LIN {X 0,Y 530.553,Z 620.523,A -85,B 0,C 180,E1 -4403.152,E2 -4403.152} C_VEL
LIN {X 0,Y 530.515,Z 626.199,A -85,B 0,C 180,E1 -4404.678,E2 -4404.678} C_VEL
LIN {X 0,Y 530.497,Z 630.318,A -85,B 0,C 180,E1 -4406.201,E2 -4406.201} C_VEL
LIN {X 0,Y 530.409,Z 633.003,A -85,B 0,C 180,E1 -4407.721,E2 -4407.721} C_VEL
LIN {X 0,Y 530.341,Z 634.333,A -85,B 0,C 180,E1 -4409.24,E2 -4409.24} C_VEL
LIN {X 0,Y 530.341,Z 634.334,A -85,B 0,C 180,E1 -4410.758,E2 -4410.758} C_VEL
LIN {X 0,Y 530.409,Z 633.003,A -85,B 0,C 180,E1 -4412.277,E2 -4412.277} C_VEL
LIN {X 0,Y 530.496,Z 630.318,A -85,B 0,C 180,E1 -4413.797,E2 -4413.797} C_VEL
LIN {X 0,Y 530.514,Z 626.204,A -85,B 0,C 180,E1 -4415.32,E2 -4415.32} C_VEL
LIN {X 0,Y 530.572,Z 620.532,A -85,B 0,C 180,E1 -4416.846,E2 -4416.846} C_VEL
LIN {X 0,Y 530.708,Z 614.132,A -85,B 0,C 180,E1 -4418.183,E2 -4418.183} C_VEL
LIN {X 0,Y 530.928,Z 606.18,A -85,B 0,C 180,E1 -4419.523,E2 -4419.523} C_VEL
LIN {X 0,Y 531.129,Z 597.86,A -85,B 0,C 180,E1 -4420.675,E2 -4420.675} C_VEL
LIN {X 0,Y 531.452,Z 587.362,A -85,B 0,C 180,E1 -4421.878,E2 -4421.878} C_VEL
LIN {X 0,Y 531.717,Z 576.66,A -85,B 0,C 180,E1 -4422.887,E2 -4422.887} C_VEL
LIN {X 0,Y 532.08,Z 564.113,A -85,B 0,C 180,E1 -4423.85,E2 -4423.85} C_VEL
LIN {X 0,Y 532.482,Z 551.655,A -85,B 0,C 180,E1 -4424.62,E2 -4424.62} C_VEL
LIN {X 0,Y 532.81,Z 537.728,A -85,B 0,C 180,E1 -4425.295,E2 -4425.295} C_VEL
LIN {X 0,Y 533.063,Z 523.832,A -85,B 0,C 180,E1 -4425.796,E2 -4425.796} C_VEL
LIN {X 0,Y 533.146,Z 510.218,A -85,B 0,C 180,E1 -4426.137,E2 -4426.137} C_VEL
LIN {X 0,Y 531.159,Z 499.764,A -85,B 0,C 180,E1 -4426.378,E2 -4426.378} C_VEL
LIN {X 0,Y 531.354,Z 487.006,A -85,B 0,C 180,E1 -4428.907,E2 -4428.907} C_VEL
LIN {X 0,Y 531.562,Z 471.4,A -85,B 0,C 180,E1 -4431.993,E2 -4431.993} C_VEL
LIN {X 0,Y 531.756,Z 457.556,A -85,B 0,C 180,E1 -4434.81,E2 -4434.81} C_VEL
LIN {X 0,Y 532.001,Z 444.494,A -85,B 0,C 180,E1 -4437.539,E2 -4437.539} C_VEL
LIN {X 0,Y 532.22,Z 430.626,A -85,B 0,C 180,E1 -4440.5,E2 -4440.5} C_VEL
LIN {X 0,Y 532.488,Z 417.378,A -85,B 0,C 180,E1 -4443.437,E2 -4443.437} C_VEL
LIN {X 0,Y 532.955,Z 402.449,A -85,B 0,C 180,E1 -4446.868,E2 -4446.868} C_VEL
LIN {X 0,Y 533.188,Z 395.134,A -85,B 0,C 180,E1 -4448.606,E2 -4448.606} C_VEL
LIN {X 0,Y 532.7,Z 391.02,A -85,B 0,C 180,E1 -4449.645,E2 -4449.645} C_VEL
LIN {X 0,Y 531.002,Z 382.968,A -85,B 0,C 180,E1 -4451.821,E2 -4451.821} C_VEL
LIN {X 0,Y 530.982,Z 382.967,A -85,B 0,C 180,E1 -4454.546,E2 -4454.546} C_VEL
LIN {X 0,Y 530.991,Z 382.971,A -85,B 0,C 180,E1 -4457.831,E2 -4457.831} C_VEL
LIN {X 0,Y 530.998,Z 382.963,A -85,B 0,C 180,E1 -4460.558,E2 -4460.558} C_VEL
LIN {X 0,Y 530.967,Z 382.972,A -85,B 0,C 180,E1 -4463.841,E2 -4463.841} C_VEL
LIN {X 0,Y 530.991,Z 382.964,A -85,B 0,C 180,E1 -4466.493,E2 -4466.493} C_VEL
LIN {X 0,Y 530.973,Z 382.97,A -85,B 0,C 180,E1 -4469.353,E2 -4469.353} C_VEL
LIN {X 0,Y 531.008,Z 382.962,A -85,B 0,C 180,E1 -4472.404,E2 -4472.404} C_VEL
LIN {X 0,Y 530.998,Z 382.964,A -85,B 0,C 180,E1 -4474.942,E2 -4474.942} C_VEL
LIN {X 0,Y 530.961,Z 382.969,A -85,B 0,C 180,E1 -4478.246,E2 -4478.246} C_VEL
LIN {X 0,Y 530.987,Z 382.964,A -85,B 0,C 180,E1 -4480.677,E2 -4480.677} C_VEL
LIN {X 0,Y 530.984,Z 382.967,A -85,B 0,C 180,E1 -4483.071,E2 -4483.071} C_VEL
LIN {X 0,Y 531.03,Z 382.966,A -85,B 0,C 180,E1 -4485.436,E2 -4485.436} C_VEL
LIN {X 0,Y 531.036,Z 382.958,A -85,B 0,C 180,E1 -4488.55,E2 -4488.55} C_VEL
LIN {X 0,Y 531.05,Z 382.962,A -85,B 0,C 180,E1 -4491.63,E2 -4491.63} C_VEL
LIN {X 0,Y 531.115,Z 382.949,A -85,B 0,C 180,E1 -4494.685,E2 -4494.685} C_VEL
LIN {X 0,Y 531.13,Z 382.951,A -85,B 0,C 180,E1 -4497.725,E2 -4497.725} C_VEL
LIN {X 0,Y 531.146,Z 382.945,A -85,B 0,C 180,E1 -4500.758,E2 -4500.758} C_VEL
LIN {X 0,Y 531.101,Z 382.953,A -85,B 0,C 180,E1 -4503.034,E2 -4503.034} C_VEL
LIN {X 0,Y 531.075,Z 382.954,A -85,B 0,C 180,E1 -4506.077,E2 -4506.077} C_VEL
LIN {X 0,Y 531.027,Z 382.965,A -85,B 0,C 180,E1 -4509.138,E2 -4509.138} C_VEL
LIN {X 0,Y 531.031,Z 382.959,A -85,B 0,C 180,E1 -4512.225,E2 -4512.225} C_VEL
LIN {X 0,Y 530.987,Z 382.971,A -85,B 0,C 180,E1 -4515.35,E2 -4515.35} C_VEL
LIN {X 0,Y 531.007,Z 382.966,A -85,B 0,C 180,E1 -4517.723,E2 -4517.723} C_VEL
LIN {X 0,Y 530.993,Z 382.967,A -85,B 0,C 180,E1 -4520.938,E2 -4520.938} C_VEL
LIN {X 0,Y 530.971,Z 382.966,A -85,B 0,C 180,E1 -4524.225,E2 -4524.225} C_VEL
LIN {X 0,Y 531.004,Z 382.964,A -85,B 0,C 180,E1 -4526.744,E2 -4526.744} C_VEL
LIN {X 0,Y 530.975,Z 382.971,A -85,B 0,C 180,E1 -4529.323,E2 -4529.323} C_VEL
LIN {X 0,Y 530.973,Z 382.966,A -85,B 0,C 180,E1 -4532.104,E2 -4532.104} C_VEL
LIN {X 0,Y 530.984,Z 382.969,A -85,B 0,C 180,E1 -4534.855,E2 -4534.855} C_VEL
LIN {X 0,Y 530.961,Z 382.972,A -85,B 0,C 180,E1 -4537.509,E2 -4537.509} C_VEL
LIN {X 0,Y 530.979,Z 382.966,A -85,B 0,C 180,E1 -4540.434,E2 -4540.434} C_VEL
LIN {X 0,Y 530.963,Z 382.972,A -85,B 0,C 180,E1 -4543.495,E2 -4543.495} C_VEL
LIN {X 0,Y 530.96,Z 382.971,A -85,B 0,C 180,E1 -4543.578,E2 -4543.578} C_VEL
LIN {X 0,Y 530.286,Z 383.052,A -85,B 0,C 180,E1 -4544.212,E2 -4544.212} C_VEL
LIN {X 0,Y 527.437,Z 383.412,A -85,B 0,C 180,E1 -4545.24,E2 -4545.24} C_VEL
LIN {X 0,Y 525.032,Z 383.714,A -85,B 0,C 180,E1 -4546.069,E2 -4546.069} C_VEL
LIN {X 0,Y 524,Z 383.84,A -85,B 0,C 180,E1 -4546.708,E2 -4546.708} C_VEL
LIN {X 0,Y 523.915,Z 383.85,A -85,B 0,C 180,E1 -4546.925,E2 -4546.925} C_VEL
LIN {X 0,Y 523.975,Z 383.838,A -85,B 0,C 180,E1 -4549.925,E2 -4549.925} C_VEL
LIN {X 0,Y 523.909,Z 383.852,A -85,B 0,C 180,E1 -4552.87,E2 -4552.87} C_VEL
LIN {X 0,Y 523.943,Z 383.843,A -85,B 0,C 180,E1 -4555.712,E2 -4555.712} C_VEL
LIN {X 0,Y 523.93,Z 383.845,A -85,B 0,C 180,E1 -4558.458,E2 -4558.458} C_VEL
LIN {X 0,Y 523.939,Z 383.847,A -85,B 0,C 180,E1 -4561.127,E2 -4561.127} C_VEL
LIN {X 0,Y 523.985,Z 383.837,A -85,B 0,C 180,E1 -4563.981,E2 -4563.981} C_VEL
LIN {X 0,Y 523.927,Z 383.845,A -85,B 0,C 180,E1 -4566.271,E2 -4566.271} C_VEL
LIN {X 0,Y 523.947,Z 383.848,A -85,B 0,C 180,E1 -4568.768,E2 -4568.768} C_VEL
LIN {X 0,Y 523.951,Z 383.845,A -85,B 0,C 180,E1 -4571.222,E2 -4571.222} C_VEL
LIN {X 0,Y 523.923,Z 383.845,A -85,B 0,C 180,E1 -4573.639,E2 -4573.639} C_VEL
LIN {X 0,Y 523.811,Z 383.865,A -85,B 0,C 180,E1 -4576.026,E2 -4576.026} C_VEL
LIN {X 0,Y 523.644,Z 383.885,A -85,B 0,C 180,E1 -4578.454,E2 -4578.454} C_VEL
LIN {X 0,Y 523.539,Z 383.897,A -85,B 0,C 180,E1 -4579.389,E2 -4579.389} C_VEL
LIN {X 0,Y 525.473,Z 393.055,A -85,B 0,C 180,E1 -4579.696,E2 -4579.696} C_VEL
LIN {X 0,Y 525.341,Z 405.307,A -85,B 0,C 180,E1 -4580.131,E2 -4580.131} C_VEL
LIN {X 0,Y 525.11,Z 416.338,A -85,B 0,C 180,E1 -4580.662,E2 -4580.662} C_VEL
LIN {X 0,Y 524.825,Z 427.193,A -85,B 0,C 180,E1 -4581.336,E2 -4581.336} C_VEL
LIN {X 0,Y 524.474,Z 438.244,A -85,B 0,C 180,E1 -4582.203,E2 -4582.203} C_VEL
LIN {X 0,Y 524.21,Z 447.187,A -85,B 0,C 180,E1 -4583.071,E2 -4583.071} C_VEL
LIN {X 0,Y 524.089,Z 455.344,A -85,B 0,C 180,E1 -4584.036,E2 -4584.036} C_VEL
LIN {X 0,Y 523.822,Z 463.291,A -85,B 0,C 180,E1 -4585.191,E2 -4585.191} C_VEL
LIN {X 0,Y 523.672,Z 470.642,A -85,B 0,C 180,E1 -4586.539,E2 -4586.539} C_VEL
LIN {X 0,Y 523.47,Z 475.563,A -85,B 0,C 180,E1 -4587.693,E2 -4587.693} C_VEL
LIN {X 0,Y 523.457,Z 479.343,A -85,B 0,C 180,E1 -4588.847,E2 -4588.847} C_VEL
LIN {X 0,Y 523.299,Z 482.152,A -85,B 0,C 180,E1 -4590.001,E2 -4590.001} C_VEL
LIN {X 0,Y 523.3,Z 484.416,A -85,B 0,C 180,E1 -4591.54,E2 -4591.54} C_VEL
LIN {X 0,Y 523.39,Z 485.162,A -85,B 0,C 180,E1 -4593.08,E2 -4593.08} C_VEL
LIN {X 0,Y 523.433,Z 484.927,A -85,B 0,C 180,E1 -4593.85,E2 -4593.85} C_VEL
LIN {X 0,Y 523.397,Z 483.363,A -85,B 0,C 180,E1 -4595.394,E2 -4595.394} C_VEL
LIN {X 0,Y 523.432,Z 481.253,A -85,B 0,C 180,E1 -4596.492,E2 -4596.492} C_VEL
LIN {X 0,Y 523.451,Z 477.911,A -85,B 0,C 180,E1 -4597.717,E2 -4597.717} C_VEL
LIN {X 0,Y 523.576,Z 473.64,A -85,B 0,C 180,E1 -4598.881,E2 -4598.881} C_VEL
LIN {X 0,Y 523.721,Z 467.117,A -85,B 0,C 180,E1 -4600.243,E2 -4600.243} C_VEL
LIN {X 0,Y 523.902,Z 459.581,A -85,B 0,C 180,E1 -4601.474,E2 -4601.474} C_VEL
LIN {X 0,Y 524.129,Z 451.055,A -85,B 0,C 180,E1 -4602.586,E2 -4602.586} C_VEL
LIN {X 0,Y 524.448,Z 440.729,A -85,B 0,C 180,E1 -4603.662,E2 -4603.662} C_VEL
LIN {X 0,Y 524.712,Z 430.134,A -85,B 0,C 180,E1 -4604.546,E2 -4604.546} C_VEL
LIN {X 0,Y 525.053,Z 418.68,A -85,B 0,C 180,E1 -4605.295,E2 -4605.295} C_VEL
LIN {X 0,Y 525.289,Z 406.308,A -85,B 0,C 180,E1 -4605.92,E2 -4605.92} C_VEL
LIN {X 0,Y 525.391,Z 392.866,A -85,B 0,C 180,E1 -4606.403,E2 -4606.403} C_VEL
LIN {X 0,Y 523.866,Z 385.46,A -85,B 0,C 180,E1 -4606.641,E2 -4606.641} C_VEL
LIN {X 0,Y 523.507,Z 383.903,A -85,B 0,C 180,E1 -4606.702,E2 -4606.702} C_VEL
LIN {X 0,Y 523.755,Z 383.871,A -85,B 0,C 180,E1 -4609.601,E2 -4609.601} C_VEL
LIN {X 0,Y 523.925,Z 383.844,A -85,B 0,C 180,E1 -4612.244,E2 -4612.244} C_VEL
LIN {X 0,Y 523.938,Z 383.844,A -85,B 0,C 180,E1 -4614.572,E2 -4614.572} C_VEL
LIN {X 0,Y 523.955,Z 383.846,A -85,B 0,C 180,E1 -4617.133,E2 -4617.133} C_VEL
LIN {X 0,Y 523.948,Z 383.842,A -85,B 0,C 180,E1 -4619.756,E2 -4619.756} C_VEL
LIN {X 0,Y 523.939,Z 383.847,A -85,B 0,C 180,E1 -4622.45,E2 -4622.45} C_VEL
LIN {X 0,Y 523.926,Z 383.846,A -85,B 0,C 180,E1 -4625.227,E2 -4625.227} C_VEL
LIN {X 0,Y 523.921,Z 383.844,A -85,B 0,C 180,E1 -4628.102,E2 -4628.102} C_VEL
LIN {X 0,Y 523.944,Z 383.842,A -85,B 0,C 180,E1 -4631.092,E2 -4631.092} C_VEL
LIN {X 0,Y 523.943,Z 383.847,A -85,B 0,C 180,E1 -4634.228,E2 -4634.228} C_VEL
LIN {X 0,Y 523.931,Z 383.845,A -85,B 0,C 180,E1 -4636.834,E2 -4636.834} C_VEL
LIN {X 0,Y 523.95,Z 383.839,A -85,B 0,C 180,E1 -4638.908,E2 -4638.908} C_VEL
LIN {X 0,Y 523.922,Z 383.839,A -85,B 0,C 180,E1 -4641.898,E2 -4641.898} C_VEL
LIN {X 0,Y 523.94,Z 383.842,A -85,B 0,C 180,E1 -4644.909,E2 -4644.909} C_VEL
LIN {X 0,Y 523.939,Z 383.845,A -85,B 0,C 180,E1 -4647.68,E2 -4647.68} C_VEL
LIN {X 0,Y 523.958,Z 383.828,A -85,B 0,C 180,E1 -4650.676,E2 -4650.676} C_VEL
LIN {X 0,Y 523.979,Z 383.841,A -85,B 0,C 180,E1 -4653.728,E2 -4653.728} C_VEL
LIN {X 0,Y 523.916,Z 383.846,A -85,B 0,C 180,E1 -4656.269,E2 -4656.269} C_VEL
LIN {X 0,Y 523.949,Z 383.841,A -85,B 0,C 180,E1 -4658.766,E2 -4658.766} C_VEL
LIN {X 0,Y 523.952,Z 383.845,A -85,B 0,C 180,E1 -4661.22,E2 -4661.22} C_VEL
LIN {X 0,Y 523.937,Z 383.849,A -85,B 0,C 180,E1 -4663.639,E2 -4663.639} C_VEL
LIN {X 0,Y 524.01,Z 383.841,A -85,B 0,C 180,E1 -4665.261,E2 -4665.261} C_VEL
LIN {X 0,Y 525.911,Z 390.795,A -85,B 0,C 180,E1 -4665.637,E2 -4665.637} C_VEL
LIN {X 0,Y 525.629,Z 403.446,A -85,B 0,C 180,E1 -4666.271,E2 -4666.271} C_VEL
LIN {X 0,Y 525.204,Z 417.065,A -85,B 0,C 180,E1 -4667.146,E2 -4667.146} C_VEL
LIN {X 0,Y 524.879,Z 428.012,A -85,B 0,C 180,E1 -4668.027,E2 -4668.027} C_VEL
LIN {X 0,Y 524.644,Z 436.155,A -85,B 0,C 180,E1 -4668.8,E2 -4668.8} C_VEL
LIN {X 0,Y 524.282,Z 444.886,A -85,B 0,C 180,E1 -4669.769,E2 -4669.769} C_VEL
LIN {X 0,Y 524.041,Z 452.329,A -85,B 0,C 180,E1 -4670.739,E2 -4670.739} C_VEL
LIN {X 0,Y 523.836,Z 458.692,A -85,B 0,C 180,E1 -4671.707,E2 -4671.707} C_VEL
LIN {X 0,Y 523.675,Z 464.14,A -85,B 0,C 180,E1 -4672.675,E2 -4672.675} C_VEL
LIN {X 0,Y 523.57,Z 469.632,A -85,B 0,C 180,E1 -4673.835,E2 -4673.835} C_VEL
LIN {X 0,Y 523.405,Z 474.136,A -85,B 0,C 180,E1 -4674.993,E2 -4674.993} C_VEL
LIN {X 0,Y 523.455,Z 477.71,A -85,B 0,C 180,E1 -4676.151,E2 -4676.151} C_VEL
LIN {X 0,Y 523.403,Z 479.714,A -85,B 0,C 180,E1 -4676.921,E2 -4676.921} C_VEL
LIN {X 0,Y 523.272,Z 482.556,A -85,B 0,C 180,E1 -4678.461,E2 -4678.461} C_VEL
LIN {X 0,Y 523.247,Z 483.583,A -85,B 0,C 180,E1 -4679.23,E2 -4679.23} C_VEL
LIN {X 0,Y 523.246,Z 484.415,A -85,B 0,C 180,E1 -4680.769,E2 -4680.769} C_VEL
LIN {X 0,Y 523.273,Z 484.415,A -85,B 0,C 180,E1 -4681.539,E2 -4681.539} C_VEL
LIN {X 0,Y 523.359,Z 483.314,A -85,B 0,C 180,E1 -4683.079,E2 -4683.079} C_VEL
LIN {X 0,Y 523.402,Z 482.253,A -85,B 0,C 180,E1 -4683.849,E2 -4683.849} C_VEL
LIN {X 0,Y 523.425,Z 479.227,A -85,B 0,C 180,E1 -4685.393,E2 -4685.393} C_VEL
LIN {X 0,Y 523.445,Z 476.197,A -85,B 0,C 180,E1 -4686.507,E2 -4686.507} C_VEL
LIN {X 0,Y 523.546,Z 470.377,A -85,B 0,C 180,E1 -4688.103,E2 -4688.103} C_VEL
LIN {X 0,Y 523.706,Z 465.027,A -85,B 0,C 180,E1 -4689.267,E2 -4689.267} C_VEL
LIN {X 0,Y 523.91,Z 458.562,A -85,B 0,C 180,E1 -4690.433,E2 -4690.433} C_VEL
LIN {X 0,Y 524.15,Z 450.803,A -85,B 0,C 180,E1 -4691.603,E2 -4691.603} C_VEL
LIN {X 0,Y 524.476,Z 441.38,A -85,B 0,C 180,E1 -4692.774,E2 -4692.774} C_VEL
LIN {X 0,Y 524.843,Z 430.786,A -85,B 0,C 180,E1 -4693.849,E2 -4693.849} C_VEL
LIN {X 0,Y 525.117,Z 421.559,A -85,B 0,C 180,E1 -4694.632,E2 -4694.632} C_VEL
LIN {X 0,Y 525.463,Z 410.674,A -85,B 0,C 180,E1 -4695.409,E2 -4695.409} C_VEL
LIN {X 0,Y 525.847,Z 398.723,A -85,B 0,C 180,E1 -4696.1,E2 -4696.1} C_VEL
LIN {X 0,Y 525.834,Z 390.325,A -85,B 0,C 180,E1 -4696.5,E2 -4696.5} C_VEL
LIN {X 0,Y 523.967,Z 383.859,A -85,B 0,C 180,E1 -4696.836,E2 -4696.836} C_VEL
LIN {X 0,Y 523.982,Z 383.844,A -85,B 0,C 180,E1 -4700.134,E2 -4700.134} C_VEL
LIN {X 0,Y 523.92,Z 383.854,A -85,B 0,C 180,E1 -4702.893,E2 -4702.893} C_VEL
LIN {X 0,Y 523.956,Z 383.848,A -85,B 0,C 180,E1 -4705.418,E2 -4705.418} C_VEL
LIN {X 0,Y 523.973,Z 383.844,A -85,B 0,C 180,E1 -4707.999,E2 -4707.999} C_VEL
LIN {X 0,Y 523.947,Z 383.846,A -85,B 0,C 180,E1 -4710.854,E2 -4710.854} C_VEL
LIN {X 0,Y 523.962,Z 383.844,A -85,B 0,C 180,E1 -4713.734,E2 -4713.734} C_VEL
LIN {X 0,Y 523.906,Z 383.853,A -85,B 0,C 180,E1 -4716.401,E2 -4716.401} C_VEL
LIN {X 0,Y 523.923,Z 383.851,A -85,B 0,C 180,E1 -4719.084,E2 -4719.084} C_VEL
LIN {X 0,Y 523.958,Z 383.845,A -85,B 0,C 180,E1 -4722.118,E2 -4722.118} C_VEL
LIN {X 0,Y 523.953,Z 383.849,A -85,B 0,C 180,E1 -4725.309,E2 -4725.309} C_VEL
LIN {X 0,Y 523.962,Z 383.847,A -85,B 0,C 180,E1 -4728.689,E2 -4728.689} C_VEL
LIN {X 0,Y 523.973,Z 384.021,A -85,B 0,C 180,E1 -4730.235,E2 -4730.235} C_VEL
LIN {X 0,Y 524.924,Z 389.904,A -85,B 0,C 180,E1 -4731.748,E2 -4731.748} C_VEL
LIN {X 0,Y 524.531,Z 400.327,A -85,B 0,C 180,E1 -4734.112,E2 -4734.112} C_VEL
LIN {X 0,Y 524.45,Z 415.646,A -85,B 0,C 180,E1 -4737.358,E2 -4737.358} C_VEL
LIN {X 0,Y 524.539,Z 431.593,A -85,B 0,C 180,E1 -4740.563,E2 -4740.563} C_VEL
LIN {X 0,Y 524.498,Z 448.042,A -85,B 0,C 180,E1 -4743.756,E2 -4743.756} C_VEL
LIN {X 0,Y 524.469,Z 463.53,A -85,B 0,C 180,E1 -4746.714,E2 -4746.714} C_VEL
LIN {X 0,Y 524.306,Z 479.649,A -85,B 0,C 180,E1 -4749.769,E2 -4749.769} C_VEL
LIN {X 0,Y 524.203,Z 494.065,A -85,B 0,C 180,E1 -4752.5,E2 -4752.5} C_VEL
LIN {X 0,Y 524.102,Z 498.948,A -85,B 0,C 180,E1 -4753.418,E2 -4753.418} C_VEL
LIN {X 0,Y 526.4,Z 512.324,A -85,B 0,C 180,E1 -4753.717,E2 -4753.717} C_VEL
LIN {X 0,Y 526.093,Z 526.732,A -85,B 0,C 180,E1 -4754.105,E2 -4754.105} C_VEL
LIN {X 0,Y 525.824,Z 540.745,A -85,B 0,C 180,E1 -4754.644,E2 -4754.644} C_VEL
LIN {X 0,Y 525.541,Z 553.328,A -85,B 0,C 180,E1 -4755.28,E2 -4755.28} C_VEL
LIN {X 0,Y 525.121,Z 565.512,A -85,B 0,C 180,E1 -4756.059,E2 -4756.059} C_VEL
LIN {X 0,Y 524.733,Z 577.736,A -85,B 0,C 180,E1 -4757.035,E2 -4757.035} C_VEL
LIN {X 0,Y 524.397,Z 588.243,A -85,B 0,C 180,E1 -4758.056,E2 -4758.056} C_VEL
LIN {X 0,Y 524.117,Z 597.847,A -85,B 0,C 180,E1 -4759.179,E2 -4759.179} C_VEL
LIN {X 0,Y 523.863,Z 606.17,A -85,B 0,C 180,E1 -4760.345,E2 -4760.345} C_VEL
LIN {X 0,Y 523.665,Z 614.123,A -85,B 0,C 180,E1 -4761.704,E2 -4761.704} C_VEL
LIN {X 0,Y 523.486,Z 620.523,A -85,B 0,C 180,E1 -4763.059,E2 -4763.059} C_VEL
LIN {X 0,Y 523.452,Z 626.199,A -85,B 0,C 180,E1 -4764.606,E2 -4764.606} C_VEL
LIN {X 0,Y 523.419,Z 630.318,A -85,B 0,C 180,E1 -4766.15,E2 -4766.15} C_VEL
LIN {X 0,Y 523.333,Z 633.004,A -85,B 0,C 180,E1 -4767.69,E2 -4767.69} C_VEL
LIN {X 0,Y 523.247,Z 634.334,A -85,B 0,C 180,E1 -4769.23,E2 -4769.23} C_VEL
LIN {X 0,Y 523.247,Z 634.334,A -85,B 0,C 180,E1 -4770.769,E2 -4770.769} C_VEL
LIN {X 0,Y 523.333,Z 633.004,A -85,B 0,C 180,E1 -4772.308,E2 -4772.308} C_VEL
LIN {X 0,Y 523.418,Z 630.318,A -85,B 0,C 180,E1 -4773.849,E2 -4773.849} C_VEL
LIN {X 0,Y 523.452,Z 626.203,A -85,B 0,C 180,E1 -4775.392,E2 -4775.392} C_VEL
LIN {X 0,Y 523.494,Z 620.532,A -85,B 0,C 180,E1 -4776.939,E2 -4776.939} C_VEL
LIN {X 0,Y 523.663,Z 614.131,A -85,B 0,C 180,E1 -4778.294,E2 -4778.294} C_VEL
LIN {X 0,Y 523.863,Z 606.18,A -85,B 0,C 180,E1 -4779.653,E2 -4779.653} C_VEL
LIN {X 0,Y 524.116,Z 597.859,A -85,B 0,C 180,E1 -4780.819,E2 -4780.819} C_VEL
LIN {X 0,Y 524.447,Z 587.098,A -85,B 0,C 180,E1 -4782.067,E2 -4782.067} C_VEL
LIN {X 0,Y 524.77,Z 576.662,A -85,B 0,C 180,E1 -4783.061,E2 -4783.061} C_VEL
LIN {X 0,Y 525.168,Z 564.111,A -85,B 0,C 180,E1 -4784.036,E2 -4784.036} C_VEL
LIN {X 0,Y 525.594,Z 551.572,A -85,B 0,C 180,E1 -4784.816,E2 -4784.816} C_VEL
LIN {X 0,Y 525.908,Z 538.563,A -85,B 0,C 180,E1 -4785.451,E2 -4785.451} C_VEL
LIN {X 0,Y 526.17,Z 524.48,A -85,B 0,C 180,E1 -4785.971,E2 -4785.971} C_VEL
LIN {X 0,Y 526.363,Z 511.554,A -85,B 0,C 180,E1 -4786.307,E2 -4786.307} C_VEL
LIN {X 0,Y 524.091,Z 499.154,A -85,B 0,C 180,E1 -4786.605,E2 -4786.605} C_VEL
LIN {X 0,Y 524.307,Z 486.266,A -85,B 0,C 180,E1 -4789.171,E2 -4789.171} C_VEL
LIN {X 0,Y 524.538,Z 470.126,A -85,B 0,C 180,E1 -4792.408,E2 -4792.408} C_VEL
LIN {X 0,Y 524.78,Z 455.935,A -85,B 0,C 180,E1 -4795.375,E2 -4795.375} C_VEL
LIN {X 0,Y 525.002,Z 442.856,A -85,B 0,C 180,E1 -4798.155,E2 -4798.155} C_VEL
LIN {X 0,Y 525.295,Z 430.576,A -85,B 0,C 180,E1 -4800.831,E2 -4800.831} C_VEL
LIN {X 0,Y 525.552,Z 418.215,A -85,B 0,C 180,E1 -4803.624,E2 -4803.624} C_VEL
LIN {X 0,Y 526.066,Z 403.921,A -85,B 0,C 180,E1 -4806.953,E2 -4806.953} C_VEL
LIN {X 0,Y 526.265,Z 395.956,A -85,B 0,C 180,E1 -4808.876,E2 -4808.876} C_VEL
LIN {X 0,Y 525.034,Z 388.915,A -85,B 0,C 180,E1 -4810.723,E2 -4810.723} C_VEL
LIN {X 0,Y 523.953,Z 383.847,A -85,B 0,C 180,E1 -4812.117,E2 -4812.117} C_VEL
LIN {X 0,Y 523.949,Z 383.845,A -85,B 0,C 180,E1 -4815.308,E2 -4815.308} C_VEL
LIN {X 0,Y 523.974,Z 383.838,A -85,B 0,C 180,E1 -4818.686,E2 -4818.686} C_VEL
LIN {X 0,Y 523.946,Z 383.842,A -85,B 0,C 180,E1 -4821.075,E2 -4821.075} C_VEL
LIN {X 0,Y 523.921,Z 383.85,A -85,B 0,C 180,E1 -4823.827,E2 -4823.827} C_VEL
LIN {X 0,Y 523.935,Z 383.843,A -85,B 0,C 180,E1 -4826.635,E2 -4826.635} C_VEL
LIN {X 0,Y 523.954,Z 383.845,A -85,B 0,C 180,E1 -4829.356,E2 -4829.356} C_VEL
LIN {X 0,Y 523.971,Z 383.84,A -85,B 0,C 180,E1 -4832.28,E2 -4832.28} C_VEL
LIN {X 0,Y 523.945,Z 383.842,A -85,B 0,C 180,E1 -4834.581,E2 -4834.581} C_VEL
LIN {X 0,Y 523.907,Z 383.849,A -85,B 0,C 180,E1 -4837.106,E2 -4837.106} C_VEL
LIN {X 0,Y 523.968,Z 383.843,A -85,B 0,C 180,E1 -4839.865,E2 -4839.865} C_VEL
LIN {X 0,Y 523.961,Z 383.84,A -85,B 0,C 180,E1 -4842.837,E2 -4842.837} C_VEL
LIN {X 0,Y 523.993,Z 383.84,A -85,B 0,C 180,E1 -4845.236,E2 -4845.236} C_VEL
LIN {X 0,Y 524.001,Z 383.835,A -85,B 0,C 180,E1 -4848.394,E2 -4848.394} C_VEL
LIN {X 0,Y 523.998,Z 383.841,A -85,B 0,C 180,E1 -4851.516,E2 -4851.516} C_VEL
LIN {X 0,Y 524.076,Z 383.825,A -85,B 0,C 180,E1 -4854.614,E2 -4854.614} C_VEL
LIN {X 0,Y 524.102,Z 383.827,A -85,B 0,C 180,E1 -4857.695,E2 -4857.695} C_VEL
LIN {X 0,Y 524.116,Z 383.821,A -85,B 0,C 180,E1 -4860.769,E2 -4860.769} C_VEL
LIN {X 0,Y 524.067,Z 383.83,A -85,B 0,C 180,E1 -4863.075,E2 -4863.075} C_VEL
LIN {X 0,Y 524.037,Z 383.831,A -85,B 0,C 180,E1 -4866.159,E2 -4866.159} C_VEL
LIN {X 0,Y 523.995,Z 383.843,A -85,B 0,C 180,E1 -4869.262,E2 -4869.262} C_VEL
LIN {X 0,Y 524.014,Z 383.837,A -85,B 0,C 180,E1 -4871.752,E2 -4871.752} C_VEL
LIN {X 0,Y 523.982,Z 383.842,A -85,B 0,C 180,E1 -4875.053,E2 -4875.053} C_VEL
LIN {X 0,Y 523.955,Z 383.842,A -85,B 0,C 180,E1 -4877.97,E2 -4877.97} C_VEL
LIN {X 0,Y 523.963,Z 383.839,A -85,B 0,C 180,E1 -4880.411,E2 -4880.411} C_VEL
LIN {X 0,Y 523.908,Z 383.85,A -85,B 0,C 180,E1 -4882.894,E2 -4882.894} C_VEL
LIN {X 0,Y 523.947,Z 383.846,A -85,B 0,C 180,E1 -4885.419,E2 -4885.419} C_VEL
LIN {X 0,Y 523.963,Z 383.84,A -85,B 0,C 180,E1 -4888,E2 -4888} C_VEL
LIN {X 0,Y 523.939,Z 383.846,A -85,B 0,C 180,E1 -4890.856,E2 -4890.856} C_VEL
LIN {X 0,Y 523.956,Z 383.843,A -85,B 0,C 180,E1 -4893.736,E2 -4893.736} C_VEL
LIN {X 0,Y 523.916,Z 383.846,A -85,B 0,C 180,E1 -4896.405,E2 -4896.405} C_VEL
LIN {X 0,Y 523.918,Z 383.852,A -85,B 0,C 180,E1 -4899.085,E2 -4899.085} C_VEL
LIN {X 0,Y 523.953,Z 383.841,A -85,B 0,C 180,E1 -4902.119,E2 -4902.119} C_VEL
LIN {X 0,Y 523.952,Z 383.846,A -85,B 0,C 180,E1 -4905.31,E2 -4905.31} C_VEL
LIN {X 0,Y 523.915,Z 383.85,A -85,B 0,C 180,E1 -4906.925,E2 -4906.925} C_VEL
LIN {X 0,Y 523.252,Z 383.931,A -85,B 0,C 180,E1 -4907.567,E2 -4907.567} C_VEL
LIN {X 0,Y 520.418,Z 384.284,A -85,B 0,C 180,E1 -4908.609,E2 -4908.609} C_VEL
LIN {X 0,Y 518.022,Z 384.584,A -85,B 0,C 180,E1 -4909.448,E2 -4909.448} C_VEL
LIN {X 0,Y 516.992,Z 384.708,A -85,B 0,C 180,E1 -4910.095,E2 -4910.095} C_VEL
LIN {X 0,Y 516.907,Z 384.719,A -85,B 0,C 180,E1 -4910.315,E2 -4910.315} C_VEL
LIN {X 0,Y 516.883,Z 384.726,A -85,B 0,C 180,E1 -4913.343,E2 -4913.343} C_VEL
LIN {X 0,Y 516.911,Z 384.718,A -85,B 0,C 180,E1 -4916.122,E2 -4916.122} C_VEL
LIN {X 0,Y 516.892,Z 384.727,A -85,B 0,C 180,E1 -4918.937,E2 -4918.937} C_VEL
LIN {X 0,Y 516.919,Z 384.719,A -85,B 0,C 180,E1 -4921.586,E2 -4921.586} C_VEL
LIN {X 0,Y 516.932,Z 384.716,A -85,B 0,C 180,E1 -4924.212,E2 -4924.212} C_VEL
LIN {X 0,Y 516.866,Z 384.73,A -85,B 0,C 180,E1 -4926.777,E2 -4926.777} C_VEL
LIN {X 0,Y 516.941,Z 384.715,A -85,B 0,C 180,E1 -4929.733,E2 -4929.733} C_VEL
LIN {X 0,Y 516.923,Z 384.721,A -85,B 0,C 180,E1 -4932.597,E2 -4932.597} C_VEL
LIN {X 0,Y 516.876,Z 384.728,A -85,B 0,C 180,E1 -4935.029,E2 -4935.029} C_VEL
LIN {X 0,Y 516.62,Z 384.76,A -85,B 0,C 180,E1 -4938.373,E2 -4938.373} C_VEL
LIN {X 0,Y 516.506,Z 384.774,A -85,B 0,C 180,E1 -4939.218,E2 -4939.218} C_VEL
LIN {X 0,Y 518.288,Z 392.23,A -85,B 0,C 180,E1 -4939.453,E2 -4939.453} C_VEL
LIN {X 0,Y 518.562,Z 398.396,A -85,B 0,C 180,E1 -4939.656,E2 -4939.656} C_VEL
LIN {X 0,Y 518.338,Z 411.499,A -85,B 0,C 180,E1 -4940.194,E2 -4940.194} C_VEL
LIN {X 0,Y 518.068,Z 422.955,A -85,B 0,C 180,E1 -4940.829,E2 -4940.829} C_VEL
LIN {X 0,Y 517.779,Z 433.912,A -85,B 0,C 180,E1 -4941.611,E2 -4941.611} C_VEL
LIN {X 0,Y 517.449,Z 444.168,A -85,B 0,C 180,E1 -4942.521,E2 -4942.521} C_VEL
LIN {X 0,Y 517.205,Z 452.345,A -85,B 0,C 180,E1 -4943.411,E2 -4943.411} C_VEL
LIN {X 0,Y 516.969,Z 460.803,A -85,B 0,C 180,E1 -4944.54,E2 -4944.54} C_VEL
LIN {X 0,Y 516.81,Z 467.875,A -85,B 0,C 180,E1 -4945.712,E2 -4945.712} C_VEL
LIN {X 0,Y 516.62,Z 473.569,A -85,B 0,C 180,E1 -4946.882,E2 -4946.882} C_VEL
LIN {X 0,Y 516.507,Z 478.052,A -85,B 0,C 180,E1 -4948.051,E2 -4948.051} C_VEL
LIN {X 0,Y 516.355,Z 481.477,A -85,B 0,C 180,E1 -4949.221,E2 -4949.221} C_VEL
LIN {X 0,Y 516.281,Z 483.234,A -85,B 0,C 180,E1 -4950.001,E2 -4950.001} C_VEL
LIN {X 0,Y 516.296,Z 485.457,A -85,B 0,C 180,E1 -4951.561,E2 -4951.561} C_VEL
LIN {X 0,Y 516.319,Z 486.009,A -85,B 0,C 180,E1 -4952.341,E2 -4952.341} C_VEL
LIN {X 0,Y 516.363,Z 486.159,A -85,B 0,C 180,E1 -4953.122,E2 -4953.122} C_VEL
LIN {X 0,Y 516.356,Z 485.3,A -85,B 0,C 180,E1 -4954.685,E2 -4954.685} C_VEL
LIN {X 0,Y 516.385,Z 484.309,A -85,B 0,C 180,E1 -4955.468,E2 -4955.468} C_VEL
LIN {X 0,Y 516.423,Z 482.223,A -85,B 0,C 180,E1 -4956.555,E2 -4956.555} C_VEL
LIN {X 0,Y 516.454,Z 478.789,A -85,B 0,C 180,E1 -4957.822,E2 -4957.822} C_VEL
LIN {X 0,Y 516.601,Z 474.477,A -85,B 0,C 180,E1 -4959.002,E2 -4959.002} C_VEL
LIN {X 0,Y 516.773,Z 467.889,A -85,B 0,C 180,E1 -4960.382,E2 -4960.382} C_VEL
LIN {X 0,Y 516.952,Z 460.543,A -85,B 0,C 180,E1 -4961.594,E2 -4961.594} C_VEL
LIN {X 0,Y 517.189,Z 453.35,A -85,B 0,C 180,E1 -4962.558,E2 -4962.558} C_VEL
LIN {X 0,Y 517.426,Z 444.376,A -85,B 0,C 180,E1 -4963.551,E2 -4963.551} C_VEL
LIN {X 0,Y 517.751,Z 434.386,A -85,B 0,C 180,E1 -4964.444,E2 -4964.444} C_VEL
LIN {X 0,Y 518.07,Z 423.583,A -85,B 0,C 180,E1 -4965.221,E2 -4965.221} C_VEL
LIN {X 0,Y 518.35,Z 411.739,A -85,B 0,C 180,E1 -4965.886,E2 -4965.886} C_VEL
LIN {X 0,Y 518.56,Z 399.112,A -85,B 0,C 180,E1 -4966.41,E2 -4966.41} C_VEL
LIN {X 0,Y 518.256,Z 392.153,A -85,B 0,C 180,E1 -4966.641,E2 -4966.641} C_VEL
LIN {X 0,Y 516.767,Z 386.025,A -85,B 0,C 180,E1 -4966.84,E2 -4966.84} C_VEL
LIN {X 0,Y 516.482,Z 384.778,A -85,B 0,C 180,E1 -4966.885,E2 -4966.885} C_VEL
LIN {X 0,Y 516.757,Z 384.743,A -85,B 0,C 180,E1 -4970.212,E2 -4970.212} C_VEL
LIN {X 0,Y 516.872,Z 384.723,A -85,B 0,C 180,E1 -4972.39,E2 -4972.39} C_VEL
LIN {X 0,Y 516.915,Z 384.722,A -85,B 0,C 180,E1 -4974.929,E2 -4974.929} C_VEL
LIN {X 0,Y 516.931,Z 384.715,A -85,B 0,C 180,E1 -4977.905,E2 -4977.905} C_VEL
LIN {X 0,Y 516.898,Z 384.721,A -85,B 0,C 180,E1 -4980.204,E2 -4980.204} C_VEL
LIN {X 0,Y 516.887,Z 384.728,A -85,B 0,C 180,E1 -4982.948,E2 -4982.948} C_VEL
LIN {X 0,Y 516.877,Z 384.723,A -85,B 0,C 180,E1 -4985.78,E2 -4985.78} C_VEL
LIN {X 0,Y 516.886,Z 384.724,A -85,B 0,C 180,E1 -4988.716,E2 -4988.716} C_VEL
LIN {X 0,Y 516.917,Z 384.717,A -85,B 0,C 180,E1 -4991.775,E2 -4991.775} C_VEL
LIN {X 0,Y 516.928,Z 384.715,A -85,B 0,C 180,E1 -4995.01,E2 -4995.01} C_VEL
LIN {X 0,Y 516.923,Z 384.72,A -85,B 0,C 180,E1 -4998.398,E2 -4998.398} C_VEL
LIN {X 0,Y 516.887,Z 384.71,A -85,B 0,C 180,E1 -5001.284,E2 -5001.284} C_VEL
LIN {X 0,Y 516.894,Z 384.726,A -85,B 0,C 180,E1 -5004.221,E2 -5004.221} C_VEL
LIN {X 0,Y 516.899,Z 384.717,A -85,B 0,C 180,E1 -5007.053,E2 -5007.053} C_VEL
LIN {X 0,Y 516.896,Z 384.713,A -85,B 0,C 180,E1 -5009.796,E2 -5009.796} C_VEL
LIN {X 0,Y 516.932,Z 384.711,A -85,B 0,C 180,E1 -5012.467,E2 -5012.467} C_VEL
LIN {X 0,Y 516.879,Z 384.722,A -85,B 0,C 180,E1 -5015.07,E2 -5015.07} C_VEL
LIN {X 0,Y 516.873,Z 384.73,A -85,B 0,C 180,E1 -5017.621,E2 -5017.621} C_VEL
LIN {X 0,Y 516.935,Z 384.716,A -85,B 0,C 180,E1 -5020.13,E2 -5020.13} C_VEL
LIN {X 0,Y 516.911,Z 384.719,A -85,B 0,C 180,E1 -5022.595,E2 -5022.595} C_VEL
LIN {X 0,Y 516.979,Z 384.716,A -85,B 0,C 180,E1 -5025.056,E2 -5025.056} C_VEL
LIN {X 0,Y 519.017,Z 391.698,A -85,B 0,C 180,E1 -5025.442,E2 -5025.442} C_VEL
LIN {X 0,Y 518.8,Z 404.296,A -85,B 0,C 180,E1 -5026.086,E2 -5026.086} C_VEL
LIN {X 0,Y 518.347,Z 417.933,A -85,B 0,C 180,E1 -5026.973,E2 -5026.973} C_VEL
LIN {X 0,Y 518.01,Z 429.002,A -85,B 0,C 180,E1 -5027.876,E2 -5027.876} C_VEL
LIN {X 0,Y 517.665,Z 438.912,A -85,B 0,C 180,E1 -5028.845,E2 -5028.845} C_VEL
LIN {X 0,Y 517.245,Z 448.99,A -85,B 0,C 180,E1 -5030.024,E2 -5030.024} C_VEL
LIN {X 0,Y 516.929,Z 458.473,A -85,B 0,C 180,E1 -5031.399,E2 -5031.399} C_VEL
LIN {X 0,Y 516.709,Z 465.091,A -85,B 0,C 180,E1 -5032.576,E2 -5032.576} C_VEL
LIN {X 0,Y 516.584,Z 470.609,A -85,B 0,C 180,E1 -5033.751,E2 -5033.751} C_VEL
LIN {X 0,Y 516.416,Z 475.13,A -85,B 0,C 180,E1 -5034.925,E2 -5034.925} C_VEL
LIN {X 0,Y 516.441,Z 478.712,A -85,B 0,C 180,E1 -5036.098,E2 -5036.098} C_VEL
LIN {X 0,Y 516.385,Z 480.725,A -85,B 0,C 180,E1 -5036.879,E2 -5036.879} C_VEL
LIN {X 0,Y 516.242,Z 483.526,A -85,B 0,C 180,E1 -5038.44,E2 -5038.44} C_VEL
LIN {X 0,Y 516.208,Z 484.505,A -85,B 0,C 180,E1 -5039.22,E2 -5039.22} C_VEL
LIN {X 0,Y 516.207,Z 485.337,A -85,B 0,C 180,E1 -5040.78,E2 -5040.78} C_VEL
LIN {X 0,Y 516.233,Z 485.322,A -85,B 0,C 180,E1 -5041.56,E2 -5041.56} C_VEL
LIN {X 0,Y 516.33,Z 484.267,A -85,B 0,C 180,E1 -5043.121,E2 -5043.121} C_VEL
LIN {X 0,Y 516.322,Z 481.895,A -85,B 0,C 180,E1 -5044.684,E2 -5044.684} C_VEL
LIN {X 0,Y 516.433,Z 479.234,A -85,B 0,C 180,E1 -5045.858,E2 -5045.858} C_VEL
LIN {X 0,Y 516.499,Z 475.76,A -85,B 0,C 180,E1 -5047.034,E2 -5047.034} C_VEL
LIN {X 0,Y 516.591,Z 471.399,A -85,B 0,C 180,E1 -5048.213,E2 -5048.213} C_VEL
LIN {X 0,Y 516.781,Z 466.025,A -85,B 0,C 180,E1 -5049.392,E2 -5049.392} C_VEL
LIN {X 0,Y 516.995,Z 459.541,A -85,B 0,C 180,E1 -5050.575,E2 -5050.575} C_VEL
LIN {X 0,Y 517.268,Z 451.733,A -85,B 0,C 180,E1 -5051.759,E2 -5051.759} C_VEL
LIN {X 0,Y 517.613,Z 442.239,A -85,B 0,C 180,E1 -5052.946,E2 -5052.946} C_VEL
LIN {X 0,Y 518.018,Z 431.62,A -85,B 0,C 180,E1 -5054.035,E2 -5054.035} C_VEL
LIN {X 0,Y 518.365,Z 421.058,A -85,B 0,C 180,E1 -5054.928,E2 -5054.928} C_VEL
LIN {X 0,Y 518.722,Z 409.703,A -85,B 0,C 180,E1 -5055.722,E2 -5055.722} C_VEL
LIN {X 0,Y 519.137,Z 396.322,A -85,B 0,C 180,E1 -5056.466,E2 -5056.466} C_VEL
LIN {X 0,Y 519.077,Z 391.94,A -85,B 0,C 180,E1 -5056.67,E2 -5056.67} C_VEL
LIN {X 0,Y 516.941,Z 384.72,A -85,B 0,C 180,E1 -5057.072,E2 -5057.072} C_VEL
LIN {X 0,Y 516.942,Z 384.722,A -85,B 0,C 180,E1 -5060.268,E2 -5060.268} C_VEL
LIN {X 0,Y 516.876,Z 384.729,A -85,B 0,C 180,E1 -5063.223,E2 -5063.223} C_VEL
LIN {X 0,Y 516.946,Z 384.719,A -85,B 0,C 180,E1 -5066.196,E2 -5066.196} C_VEL
LIN {X 0,Y 516.924,Z 384.722,A -85,B 0,C 180,E1 -5069.304,E2 -5069.304} C_VEL
LIN {X 0,Y 516.9,Z 384.724,A -85,B 0,C 180,E1 -5072.543,E2 -5072.543} C_VEL
LIN {X 0,Y 516.869,Z 384.73,A -85,B 0,C 180,E1 -5075.329,E2 -5075.329} C_VEL
LIN {X 0,Y 516.883,Z 384.728,A -85,B 0,C 180,E1 -5077.943,E2 -5077.943} C_VEL
LIN {X 0,Y 516.887,Z 384.726,A -85,B 0,C 180,E1 -5080.741,E2 -5080.741} C_VEL
LIN {X 0,Y 516.887,Z 384.729,A -85,B 0,C 180,E1 -5082.831,E2 -5082.831} C_VEL
LIN {X 0,Y 516.926,Z 384.724,A -85,B 0,C 180,E1 -5085.01,E2 -5085.01} C_VEL
LIN {X 0,Y 516.918,Z 384.724,A -85,B 0,C 180,E1 -5088.398,E2 -5088.398} C_VEL
LIN {X 0,Y 516.929,Z 384.856,A -85,B 0,C 180,E1 -5089.97,E2 -5089.97} C_VEL
LIN {X 0,Y 517.999,Z 391.311,A -85,B 0,C 180,E1 -5091.687,E2 -5091.687} C_VEL
LIN {X 0,Y 517.566,Z 401.409,A -85,B 0,C 180,E1 -5094.035,E2 -5094.035} C_VEL
LIN {X 0,Y 517.431,Z 416.787,A -85,B 0,C 180,E1 -5097.364,E2 -5097.364} C_VEL
LIN {X 0,Y 517.47,Z 431.432,A -85,B 0,C 180,E1 -5100.367,E2 -5100.367} C_VEL
LIN {X 0,Y 517.43,Z 446.578,A -85,B 0,C 180,E1 -5103.37,E2 -5103.37} C_VEL
LIN {X 0,Y 517.394,Z 460.958,A -85,B 0,C 180,E1 -5106.164,E2 -5106.164} C_VEL
LIN {X 0,Y 517.243,Z 476.242,A -85,B 0,C 180,E1 -5109.104,E2 -5109.104} C_VEL
LIN {X 0,Y 517.117,Z 490.195,A -85,B 0,C 180,E1 -5111.784,E2 -5111.784} C_VEL
LIN {X 0,Y 517.006,Z 497.473,A -85,B 0,C 180,E1 -5113.184,E2 -5113.184} C_VEL
LIN {X 0,Y 518.356,Z 506.693,A -85,B 0,C 180,E1 -5113.384,E2 -5113.384} C_VEL
LIN {X 0,Y 519.514,Z 513.182,A -85,B 0,C 180,E1 -5113.557,E2 -5113.557} C_VEL
LIN {X 0,Y 519.128,Z 527.906,A -85,B 0,C 180,E1 -5113.988,E2 -5113.988} C_VEL
LIN {X 0,Y 518.768,Z 542.208,A -85,B 0,C 180,E1 -5114.581,E2 -5114.581} C_VEL
LIN {X 0,Y 518.477,Z 555.133,A -85,B 0,C 180,E1 -5115.276,E2 -5115.276} C_VEL
LIN {X 0,Y 518.005,Z 568.347,A -85,B 0,C 180,E1 -5116.164,E2 -5116.164} C_VEL
LIN {X 0,Y 517.633,Z 580.292,A -85,B 0,C 180,E1 -5117.154,E2 -5117.154} C_VEL
LIN {X 0,Y 517.33,Z 591.128,A -85,B 0,C 180,E1 -5118.241,E2 -5118.241} C_VEL
LIN {X 0,Y 517.002,Z 600.774,A -85,B 0,C 180,E1 -5119.425,E2 -5119.425} C_VEL
LIN {X 0,Y 516.773,Z 608.63,A -85,B 0,C 180,E1 -5120.607,E2 -5120.607} C_VEL
LIN {X 0,Y 516.577,Z 615.129,A -85,B 0,C 180,E1 -5121.786,E2 -5121.786} C_VEL
LIN {X 0,Y 516.399,Z 620.523,A -85,B 0,C 180,E1 -5122.964,E2 -5122.964} C_VEL
LIN {X 0,Y 516.388,Z 626.198,A -85,B 0,C 180,E1 -5124.532,E2 -5124.532} C_VEL
LIN {X 0,Y 516.325,Z 630.318,A -85,B 0,C 180,E1 -5126.097,E2 -5126.097} C_VEL
LIN {X 0,Y 516.259,Z 633.004,A -85,B 0,C 180,E1 -5127.659,E2 -5127.659} C_VEL
LIN {X 0,Y 516.157,Z 634.334,A -85,B 0,C 180,E1 -5129.219,E2 -5129.219} C_VEL
LIN {X 0,Y 516.157,Z 634.334,A -85,B 0,C 180,E1 -5130.779,E2 -5130.779} C_VEL
LIN {X 0,Y 516.259,Z 633.004,A -85,B 0,C 180,E1 -5132.34,E2 -5132.34} C_VEL
LIN {X 0,Y 516.324,Z 630.318,A -85,B 0,C 180,E1 -5133.902,E2 -5133.902} C_VEL
LIN {X 0,Y 516.387,Z 626.203,A -85,B 0,C 180,E1 -5135.466,E2 -5135.466} C_VEL
LIN {X 0,Y 516.405,Z 620.531,A -85,B 0,C 180,E1 -5137.035,E2 -5137.035} C_VEL
LIN {X 0,Y 516.598,Z 614.131,A -85,B 0,C 180,E1 -5138.409,E2 -5138.409} C_VEL
LIN {X 0,Y 516.826,Z 606.179,A -85,B 0,C 180,E1 -5139.786,E2 -5139.786} C_VEL
LIN {X 0,Y 517.111,Z 597.774,A -85,B 0,C 180,E1 -5140.968,E2 -5140.968} C_VEL
LIN {X 0,Y 517.422,Z 587.082,A -85,B 0,C 180,E1 -5142.197,E2 -5142.197} C_VEL
LIN {X 0,Y 517.779,Z 576.018,A -85,B 0,C 180,E1 -5143.24,E2 -5143.24} C_VEL
LIN {X 0,Y 518.191,Z 563.173,A -85,B 0,C 180,E1 -5144.229,E2 -5144.229} C_VEL
LIN {X 0,Y 518.649,Z 550.466,A -85,B 0,C 180,E1 -5145.019,E2 -5145.019} C_VEL
LIN {X 0,Y 519.023,Z 537.43,A -85,B 0,C 180,E1 -5145.661,E2 -5145.661} C_VEL
LIN {X 0,Y 519.269,Z 524.141,A -85,B 0,C 180,E1 -5146.162,E2 -5146.162} C_VEL
LIN {X 0,Y 519.426,Z 512.058,A -85,B 0,C 180,E1 -5146.493,E2 -5146.493} C_VEL
LIN {X 0,Y 517.092,Z 499.13,A -85,B 0,C 180,E1 -5146.802,E2 -5146.802} C_VEL
LIN {X 0,Y 517.062,Z 498.357,A -85,B 0,C 180,E1 -5146.838,E2 -5146.838} C_VEL
LIN {X 0,Y 517.306,Z 483.493,A -85,B 0,C 180,E1 -5149.854,E2 -5149.854} C_VEL
LIN {X 0,Y 517.537,Z 469.016,A -85,B 0,C 180,E1 -5152.829,E2 -5152.829} C_VEL
LIN {X 0,Y 517.848,Z 453.722,A -85,B 0,C 180,E1 -5156.07,E2 -5156.07} C_VEL
LIN {X 0,Y 518.132,Z 439.213,A -85,B 0,C 180,E1 -5159.228,E2 -5159.228} C_VEL
LIN {X 0,Y 518.484,Z 425.262,A -85,B 0,C 180,E1 -5162.371,E2 -5162.371} C_VEL
LIN {X 0,Y 518.885,Z 411.235,A -85,B 0,C 180,E1 -5165.643,E2 -5165.643} C_VEL
LIN {X 0,Y 519.429,Z 399.407,A -85,B 0,C 180,E1 -5168.489,E2 -5168.489} C_VEL
LIN {X 0,Y 518.921,Z 394.386,A -85,B 0,C 180,E1 -5169.783,E2 -5169.783} C_VEL
LIN {X 0,Y 516.894,Z 384.724,A -85,B 0,C 180,E1 -5172.444,E2 -5172.444} C_VEL
LIN {X 0,Y 516.915,Z 384.72,A -85,B 0,C 180,E1 -5175.009,E2 -5175.009} C_VEL
LIN {X 0,Y 516.922,Z 384.718,A -85,B 0,C 180,E1 -5178.396,E2 -5178.396} C_VEL
LIN {X 0,Y 516.898,Z 384.722,A -85,B 0,C 180,E1 -5181.286,E2 -5181.286} C_VEL
LIN {X 0,Y 516.883,Z 384.724,A -85,B 0,C 180,E1 -5184.221,E2 -5184.221} C_VEL
LIN {X 0,Y 516.889,Z 384.722,A -85,B 0,C 180,E1 -5187.053,E2 -5187.053} C_VEL
LIN {X 0,Y 516.893,Z 384.725,A -85,B 0,C 180,E1 -5189.796,E2 -5189.796} C_VEL
LIN {X 0,Y 516.921,Z 384.717,A -85,B 0,C 180,E1 -5192.467,E2 -5192.467} C_VEL
LIN {X 0,Y 516.902,Z 384.721,A -85,B 0,C 180,E1 -5195.072,E2 -5195.072} C_VEL
LIN {X 0,Y 516.876,Z 384.723,A -85,B 0,C 180,E1 -5198.462,E2 -5198.462} C_VEL
LIN {X 0,Y 516.895,Z 384.721,A -85,B 0,C 180,E1 -5200.955,E2 -5200.955} C_VEL
LIN {X 0,Y 516.908,Z 384.725,A -85,B 0,C 180,E1 -5203.41,E2 -5203.41} C_VEL
LIN {X 0,Y 516.896,Z 384.724,A -85,B 0,C 180,E1 -5205.834,E2 -5205.834} C_VEL
LIN {X 0,Y 516.993,Z 384.709,A -85,B 0,C 180,E1 -5208.234,E2 -5208.234} C_VEL
LIN {X 0,Y 516.962,Z 384.718,A -85,B 0,C 180,E1 -5211.4,E2 -5211.4} C_VEL
LIN {X 0,Y 517,Z 384.711,A -85,B 0,C 180,E1 -5213.757,E2 -5213.757} C_VEL
LIN {X 0,Y 517.008,Z 384.707,A -85,B 0,C 180,E1 -5216.883,E2 -5216.883} C_VEL
LIN {X 0,Y 517.074,Z 384.7,A -85,B 0,C 180,E1 -5220,E2 -5220} C_VEL
LIN {X 0,Y 517.008,Z 384.71,A -85,B 0,C 180,E1 -5223.117,E2 -5223.117} C_VEL
LIN {X 0,Y 517.001,Z 384.707,A -85,B 0,C 180,E1 -5226.244,E2 -5226.244} C_VEL
LIN {X 0,Y 516.949,Z 384.719,A -85,B 0,C 180,E1 -5229.39,E2 -5229.39} C_VEL
LIN {X 0,Y 516.973,Z 384.713,A -85,B 0,C 180,E1 -5231.825,E2 -5231.825} C_VEL
LIN {X 0,Y 516.934,Z 384.721,A -85,B 0,C 180,E1 -5235.147,E2 -5235.147} C_VEL
LIN {X 0,Y 516.917,Z 384.717,A -85,B 0,C 180,E1 -5238.223,E2 -5238.223} C_VEL
LIN {X 0,Y 516.904,Z 384.72,A -85,B 0,C 180,E1 -5240.702,E2 -5240.702} C_VEL
LIN {X 0,Y 516.902,Z 384.72,A -85,B 0,C 180,E1 -5244.073,E2 -5244.073} C_VEL
LIN {X 0,Y 516.921,Z 384.718,A -85,B 0,C 180,E1 -5246.658,E2 -5246.658} C_VEL
LIN {X 0,Y 516.904,Z 384.723,A -85,B 0,C 180,E1 -5249.525,E2 -5249.525} C_VEL
LIN {X 0,Y 516.894,Z 384.721,A -85,B 0,C 180,E1 -5252.545,E2 -5252.545} C_VEL
LIN {X 0,Y 516.877,Z 384.727,A -85,B 0,C 180,E1 -5255.334,E2 -5255.334} C_VEL
LIN {X 0,Y 516.876,Z 384.723,A -85,B 0,C 180,E1 -5257.944,E2 -5257.944} C_VEL
LIN {X 0,Y 516.88,Z 384.725,A -85,B 0,C 180,E1 -5260.742,E2 -5260.742} C_VEL
LIN {X 0,Y 516.9,Z 384.724,A -85,B 0,C 180,E1 -5262.83,E2 -5262.83} C_VEL
LIN {X 0,Y 516.918,Z 384.724,A -85,B 0,C 180,E1 -5265.011,E2 -5265.011} C_VEL
LIN {X 0,Y 516.919,Z 384.718,A -85,B 0,C 180,E1 -5268.399,E2 -5268.399} C_VEL
LIN {X 0,Y 516.907,Z 384.719,A -85,B 0,C 180,E1 -5270.315,E2 -5270.315} C_VEL
LIN {X 0,Y 516.238,Z 384.808,A -85,B 0,C 180,E1 -5270.965,E2 -5270.965} C_VEL
LIN {X 0,Y 513.381,Z 385.164,A -85,B 0,C 180,E1 -5272.02,E2 -5272.02} C_VEL
LIN {X 0,Y 510.962,Z 385.465,A -85,B 0,C 180,E1 -5272.87,E2 -5272.87} C_VEL
LIN {X 0,Y 509.917,Z 385.592,A -85,B 0,C 180,E1 -5273.526,E2 -5273.526} C_VEL
LIN {X 0,Y 509.829,Z 385.602,A -85,B 0,C 180,E1 -5273.749,E2 -5273.749} C_VEL
LIN {X 0,Y 509.861,Z 385.599,A -85,B 0,C 180,E1 -5276.541,E2 -5276.541} C_VEL
LIN {X 0,Y 509.845,Z 385.602,A -85,B 0,C 180,E1 -5279.336,E2 -5279.336} C_VEL
LIN {X 0,Y 509.893,Z 385.593,A -85,B 0,C 180,E1 -5282.056,E2 -5282.056} C_VEL
LIN {X 0,Y 509.877,Z 385.599,A -85,B 0,C 180,E1 -5284.705,E2 -5284.705} C_VEL
LIN {X 0,Y 509.828,Z 385.603,A -85,B 0,C 180,E1 -5287.459,E2 -5287.459} C_VEL
LIN {X 0,Y 509.918,Z 385.59,A -85,B 0,C 180,E1 -5289.846,E2 -5289.846} C_VEL
LIN {X 0,Y 509.877,Z 385.598,A -85,B 0,C 180,E1 -5293.176,E2 -5293.176} C_VEL
LIN {X 0,Y 509.773,Z 385.612,A -85,B 0,C 180,E1 -5295.633,E2 -5295.633} C_VEL
LIN {X 0,Y 509.576,Z 385.638,A -85,B 0,C 180,E1 -5298.302,E2 -5298.302} C_VEL
LIN {X 0,Y 509.513,Z 385.647,A -85,B 0,C 180,E1 -5299.018,E2 -5299.018} C_VEL
LIN {X 0,Y 511.476,Z 393.52,A -85,B 0,C 180,E1 -5299.279,E2 -5299.279} C_VEL
LIN {X 0,Y 511.726,Z 397.729,A -85,B 0,C 180,E1 -5299.416,E2 -5299.416} C_VEL
LIN {X 0,Y 511.577,Z 410.194,A -85,B 0,C 180,E1 -5299.913,E2 -5299.913} C_VEL
LIN {X 0,Y 511.275,Z 421.377,A -85,B 0,C 180,E1 -5300.507,E2 -5300.507} C_VEL
LIN {X 0,Y 510.951,Z 432.964,A -85,B 0,C 180,E1 -5301.299,E2 -5301.299} C_VEL
LIN {X 0,Y 510.627,Z 443.507,A -85,B 0,C 180,E1 -5302.218,E2 -5302.218} C_VEL
LIN {X 0,Y 510.297,Z 451.69,A -85,B 0,C 180,E1 -5303.086,E2 -5303.086} C_VEL
LIN {X 0,Y 510.121,Z 460.753,A -85,B 0,C 180,E1 -5304.268,E2 -5304.268} C_VEL
LIN {X 0,Y 509.858,Z 468.035,A -85,B 0,C 180,E1 -5305.455,E2 -5305.455} C_VEL
LIN {X 0,Y 509.639,Z 474.747,A -85,B 0,C 180,E1 -5306.839,E2 -5306.839} C_VEL
LIN {X 0,Y 509.497,Z 479.196,A -85,B 0,C 180,E1 -5308.025,E2 -5308.025} C_VEL
LIN {X 0,Y 509.361,Z 482.582,A -85,B 0,C 180,E1 -5309.21,E2 -5309.21} C_VEL
LIN {X 0,Y 509.262,Z 484.311,A -85,B 0,C 180,E1 -5310.001,E2 -5310.001} C_VEL
LIN {X 0,Y 509.29,Z 486.498,A -85,B 0,C 180,E1 -5311.582,E2 -5311.582} C_VEL
LIN {X 0,Y 509.294,Z 487.036,A -85,B 0,C 180,E1 -5312.373,E2 -5312.373} C_VEL
LIN {X 0,Y 509.368,Z 486.89,A -85,B 0,C 180,E1 -5313.957,E2 -5313.957} C_VEL
LIN {X 0,Y 509.375,Z 485.251,A -85,B 0,C 180,E1 -5315.543,E2 -5315.543} C_VEL
LIN {X 0,Y 509.409,Z 483.208,A -85,B 0,C 180,E1 -5316.612,E2 -5316.612} C_VEL
LIN {X 0,Y 509.458,Z 479.667,A -85,B 0,C 180,E1 -5317.93,E2 -5317.93} C_VEL
LIN {X 0,Y 509.633,Z 475.309,A -85,B 0,C 180,E1 -5319.126,E2 -5319.126} C_VEL
LIN {X 0,Y 509.825,Z 468.663,A -85,B 0,C 180,E1 -5320.525,E2 -5320.525} C_VEL
LIN {X 0,Y 510.018,Z 461.454,A -85,B 0,C 180,E1 -5321.725,E2 -5321.725} C_VEL
LIN {X 0,Y 510.272,Z 454.014,A -85,B 0,C 180,E1 -5322.731,E2 -5322.731} C_VEL
LIN {X 0,Y 510.561,Z 444.931,A -85,B 0,C 180,E1 -5323.737,E2 -5323.737} C_VEL
LIN {X 0,Y 510.88,Z 434.85,A -85,B 0,C 180,E1 -5324.643,E2 -5324.643} C_VEL
LIN {X 0,Y 511.224,Z 424.232,A -85,B 0,C 180,E1 -5325.409,E2 -5325.409} C_VEL
LIN {X 0,Y 511.501,Z 412.874,A -85,B 0,C 180,E1 -5326.053,E2 -5326.053} C_VEL
LIN {X 0,Y 511.712,Z 400.283,A -85,B 0,C 180,E1 -5326.584,E2 -5326.584} C_VEL
LIN {X 0,Y 511.416,Z 393.147,A -85,B 0,C 180,E1 -5326.825,E2 -5326.825} C_VEL
LIN {X 0,Y 509.45,Z 385.655,A -85,B 0,C 180,E1 -5327.073,E2 -5327.073} C_VEL
LIN {X 0,Y 509.735,Z 385.617,A -85,B 0,C 180,E1 -5330.354,E2 -5330.354} C_VEL
LIN {X 0,Y 509.828,Z 385.603,A -85,B 0,C 180,E1 -5332.705,E2 -5332.705} C_VEL
LIN {X 0,Y 509.882,Z 385.598,A -85,B 0,C 180,E1 -5335.296,E2 -5335.296} C_VEL
LIN {X 0,Y 509.902,Z 385.591,A -85,B 0,C 180,E1 -5338.101,E2 -5338.101} C_VEL
LIN {X 0,Y 509.852,Z 385.601,A -85,B 0,C 180,E1 -5341.28,E2 -5341.28} C_VEL
LIN {X 0,Y 509.849,Z 385.6,A -85,B 0,C 180,E1 -5344.2,E2 -5344.2} C_VEL
LIN {X 0,Y 509.822,Z 385.598,A -85,B 0,C 180,E1 -5347.341,E2 -5347.341} C_VEL
LIN {X 0,Y 509.843,Z 385.603,A -85,B 0,C 180,E1 -5350.382,E2 -5350.382} C_VEL
LIN {X 0,Y 509.828,Z 385.601,A -85,B 0,C 180,E1 -5353.062,E2 -5353.062} C_VEL
LIN {X 0,Y 509.836,Z 385.599,A -85,B 0,C 180,E1 -5355.792,E2 -5355.792} C_VEL
LIN {X 0,Y 509.864,Z 385.597,A -85,B 0,C 180,E1 -5358.575,E2 -5358.575} C_VEL
LIN {X 0,Y 509.857,Z 385.588,A -85,B 0,C 180,E1 -5361.786,E2 -5361.786} C_VEL
LIN {X 0,Y 509.849,Z 385.599,A -85,B 0,C 180,E1 -5364.623,E2 -5364.623} C_VEL
LIN {X 0,Y 509.866,Z 385.596,A -85,B 0,C 180,E1 -5367.481,E2 -5367.481} C_VEL
LIN {X 0,Y 509.863,Z 385.585,A -85,B 0,C 180,E1 -5370.274,E2 -5370.274} C_VEL
LIN {X 0,Y 509.889,Z 385.587,A -85,B 0,C 180,E1 -5372.944,E2 -5372.944} C_VEL
LIN {X 0,Y 509.855,Z 385.602,A -85,B 0,C 180,E1 -5375.573,E2 -5375.573} C_VEL
LIN {X 0,Y 509.825,Z 385.602,A -85,B 0,C 180,E1 -5378.148,E2 -5378.148} C_VEL
LIN {X 0,Y 509.866,Z 385.595,A -85,B 0,C 180,E1 -5380.681,E2 -5380.681} C_VEL
LIN {X 0,Y 509.879,Z 385.6,A -85,B 0,C 180,E1 -5383.174,E2 -5383.174} C_VEL
LIN {X 0,Y 509.926,Z 385.723,A -85,B 0,C 180,E1 -5384.864,E2 -5384.864} C_VEL
LIN {X 0,Y 512.277,Z 393.676,A -85,B 0,C 180,E1 -5385.297,E2 -5385.297} C_VEL
LIN {X 0,Y 511.924,Z 406.877,A -85,B 0,C 180,E1 -5385.997,E2 -5385.997} C_VEL
LIN {X 0,Y 511.499,Z 418.798,A -85,B 0,C 180,E1 -5386.795,E2 -5386.795} C_VEL
LIN {X 0,Y 511.122,Z 429.999,A -85,B 0,C 180,E1 -5387.72,E2 -5387.72} C_VEL
LIN {X 0,Y 510.775,Z 439.812,A -85,B 0,C 180,E1 -5388.692,E2 -5388.692} C_VEL
LIN {X 0,Y 510.309,Z 449.895,A -85,B 0,C 180,E1 -5389.887,E2 -5389.887} C_VEL
LIN {X 0,Y 509.98,Z 459.395,A -85,B 0,C 180,E1 -5391.281,E2 -5391.281} C_VEL
LIN {X 0,Y 509.741,Z 466.043,A -85,B 0,C 180,E1 -5392.474,E2 -5392.474} C_VEL
LIN {X 0,Y 509.598,Z 471.587,A -85,B 0,C 180,E1 -5393.665,E2 -5393.665} C_VEL
LIN {X 0,Y 509.427,Z 476.125,A -85,B 0,C 180,E1 -5394.855,E2 -5394.855} C_VEL
LIN {X 0,Y 509.428,Z 479.714,A -85,B 0,C 180,E1 -5396.044,E2 -5396.044} C_VEL
LIN {X 0,Y 509.366,Z 481.719,A -85,B 0,C 180,E1 -5396.836,E2 -5396.836} C_VEL
LIN {X 0,Y 509.241,Z 484.558,A -85,B 0,C 180,E1 -5398.418,E2 -5398.418} C_VEL
LIN {X 0,Y 509.198,Z 485.519,A -85,B 0,C 180,E1 -5399.209,E2 -5399.209} C_VEL
LIN {X 0,Y 509.196,Z 486.388,A -85,B 0,C 180,E1 -5400.791,E2 -5400.791} C_VEL
LIN {X 0,Y 509.279,Z 485.959,A -85,B 0,C 180,E1 -5402.373,E2 -5402.373} C_VEL
LIN {X 0,Y 509.362,Z 484.292,A -85,B 0,C 180,E1 -5403.956,E2 -5403.956} C_VEL
LIN {X 0,Y 509.472,Z 481.286,A -85,B 0,C 180,E1 -5405.541,E2 -5405.541} C_VEL
LIN {X 0,Y 509.52,Z 476.794,A -85,B 0,C 180,E1 -5407.131,E2 -5407.131} C_VEL
LIN {X 0,Y 509.635,Z 472.422,A -85,B 0,C 180,E1 -5408.325,E2 -5408.325} C_VEL
LIN {X 0,Y 509.847,Z 466.048,A -85,B 0,C 180,E1 -5409.721,E2 -5409.721} C_VEL
LIN {X 0,Y 510.151,Z 458.076,A -85,B 0,C 180,E1 -5411.12,E2 -5411.12} C_VEL
LIN {X 0,Y 510.478,Z 449.984,A -85,B 0,C 180,E1 -5412.281,E2 -5412.281} C_VEL
LIN {X 0,Y 510.809,Z 441.334,A -85,B 0,C 180,E1 -5413.324,E2 -5413.324} C_VEL
LIN {X 0,Y 511.216,Z 431.375,A -85,B 0,C 180,E1 -5414.327,E2 -5414.327} C_VEL
LIN {X 0,Y 511.618,Z 420.658,A -85,B 0,C 180,E1 -5415.224,E2 -5415.224} C_VEL
LIN {X 0,Y 511.978,Z 408.154,A -85,B 0,C 180,E1 -5416.074,E2 -5416.074} C_VEL
LIN {X 0,Y 512.391,Z 394.63,A -85,B 0,C 180,E1 -5416.792,E2 -5416.792} C_VEL
LIN {X 0,Y 511.39,Z 390.685,A -85,B 0,C 180,E1 -5417.012,E2 -5417.012} C_VEL
LIN {X 0,Y 509.888,Z 385.599,A -85,B 0,C 180,E1 -5417.29,E2 -5417.29} C_VEL
LIN {X 0,Y 509.889,Z 385.601,A -85,B 0,C 180,E1 -5420.401,E2 -5420.401} C_VEL
LIN {X 0,Y 509.84,Z 385.605,A -85,B 0,C 180,E1 -5423.563,E2 -5423.563} C_VEL
LIN {X 0,Y 509.915,Z 385.597,A -85,B 0,C 180,E1 -5426.378,E2 -5426.378} C_VEL
LIN {X 0,Y 509.88,Z 385.598,A -85,B 0,C 180,E1 -5428.844,E2 -5428.844} C_VEL
LIN {X 0,Y 509.824,Z 385.607,A -85,B 0,C 180,E1 -5431.59,E2 -5431.59} C_VEL
LIN {X 0,Y 509.85,Z 385.603,A -85,B 0,C 180,E1 -5434.413,E2 -5434.413} C_VEL
LIN {X 0,Y 509.819,Z 385.606,A -85,B 0,C 180,E1 -5437.341,E2 -5437.341} C_VEL
LIN {X 0,Y 509.841,Z 385.605,A -85,B 0,C 180,E1 -5440.382,E2 -5440.382} C_VEL
LIN {X 0,Y 509.827,Z 385.606,A -85,B 0,C 180,E1 -5443.062,E2 -5443.062} C_VEL
LIN {X 0,Y 509.833,Z 385.607,A -85,B 0,C 180,E1 -5445.792,E2 -5445.792} C_VEL
LIN {X 0,Y 509.86,Z 385.604,A -85,B 0,C 180,E1 -5448.574,E2 -5448.574} C_VEL
LIN {X 0,Y 509.873,Z 385.652,A -85,B 0,C 180,E1 -5449.676,E2 -5449.676} C_VEL
LIN {X 0,Y 511.078,Z 392.666,A -85,B 0,C 180,E1 -5451.612,E2 -5451.612} C_VEL
LIN {X 0,Y 510.588,Z 402.942,A -85,B 0,C 180,E1 -5454.055,E2 -5454.055} C_VEL
LIN {X 0,Y 510.387,Z 418.635,A -85,B 0,C 180,E1 -5457.518,E2 -5457.518} C_VEL
LIN {X 0,Y 510.426,Z 432.978,A -85,B 0,C 180,E1 -5460.512,E2 -5460.512} C_VEL
LIN {X 0,Y 510.35,Z 447.92,A -85,B 0,C 180,E1 -5463.523,E2 -5463.523} C_VEL
LIN {X 0,Y 510.305,Z 462.793,A -85,B 0,C 180,E1 -5466.459,E2 -5466.459} C_VEL
LIN {X 0,Y 510.136,Z 478.489,A -85,B 0,C 180,E1 -5469.524,E2 -5469.524} C_VEL
LIN {X 0,Y 510.007,Z 494.069,A -85,B 0,C 180,E1 -5472.559,E2 -5472.559} C_VEL
LIN {X 0,Y 509.949,Z 496.045,A -85,B 0,C 180,E1 -5472.944,E2 -5472.944} C_VEL
LIN {X 0,Y 511.25,Z 506.463,A -85,B 0,C 180,E1 -5473.183,E2 -5473.183} C_VEL
LIN {X 0,Y 512.544,Z 514.3,A -85,B 0,C 180,E1 -5473.406,E2 -5473.406} C_VEL
LIN {X 0,Y 512.171,Z 528.358,A -85,B 0,C 180,E1 -5473.85,E2 -5473.85} C_VEL
LIN {X 0,Y 511.755,Z 542.548,A -85,B 0,C 180,E1 -5474.466,E2 -5474.466} C_VEL
LIN {X 0,Y 511.451,Z 555.139,A -85,B 0,C 180,E1 -5475.17,E2 -5475.17} C_VEL
LIN {X 0,Y 510.99,Z 566.8,A -85,B 0,C 180,E1 -5475.971,E2 -5475.971} C_VEL
LIN {X 0,Y 510.609,Z 578.817,A -85,B 0,C 180,E1 -5476.974,E2 -5476.974} C_VEL
LIN {X 0,Y 510.263,Z 589.721,A -85,B 0,C 180,E1 -5478.076,E2 -5478.076} C_VEL
LIN {X 0,Y 509.959,Z 599.58,A -85,B 0,C 180,E1 -5479.277,E2 -5479.277} C_VEL
LIN {X 0,Y 509.674,Z 608.974,A -85,B 0,C 180,E1 -5480.675,E2 -5480.675} C_VEL
LIN {X 0,Y 509.425,Z 616.535,A -85,B 0,C 180,E1 -5482.069,E2 -5482.069} C_VEL
LIN {X 0,Y 509.308,Z 622.666,A -85,B 0,C 180,E1 -5483.482,E2 -5483.482} C_VEL
LIN {X 0,Y 509.239,Z 627.27,A -85,B 0,C 180,E1 -5484.852,E2 -5484.852} C_VEL
LIN {X 0,Y 509.218,Z 630.273,A -85,B 0,C 180,E1 -5486.042,E2 -5486.042} C_VEL
LIN {X 0,Y 509.159,Z 632.992,A -85,B 0,C 180,E1 -5487.626,E2 -5487.626} C_VEL
LIN {X 0,Y 509.071,Z 634.33,A -85,B 0,C 180,E1 -5489.208,E2 -5489.208} C_VEL
LIN {X 0,Y 509.071,Z 634.33,A -85,B 0,C 180,E1 -5490.79,E2 -5490.79} C_VEL
LIN {X 0,Y 509.158,Z 632.992,A -85,B 0,C 180,E1 -5492.372,E2 -5492.372} C_VEL
LIN {X 0,Y 509.218,Z 630.273,A -85,B 0,C 180,E1 -5493.956,E2 -5493.956} C_VEL
LIN {X 0,Y 509.299,Z 626.065,A -85,B 0,C 180,E1 -5495.542,E2 -5495.542} C_VEL
LIN {X 0,Y 509.337,Z 622.01,A -85,B 0,C 180,E1 -5496.695,E2 -5496.695} C_VEL
LIN {X 0,Y 509.423,Z 616.586,A -85,B 0,C 180,E1 -5497.929,E2 -5497.929} C_VEL
LIN {X 0,Y 509.668,Z 609.093,A -85,B 0,C 180,E1 -5499.323,E2 -5499.323} C_VEL
LIN {X 0,Y 509.958,Z 599.817,A -85,B 0,C 180,E1 -5500.721,E2 -5500.721} C_VEL
LIN {X 0,Y 510.232,Z 590.095,A -85,B 0,C 180,E1 -5501.923,E2 -5501.923} C_VEL
LIN {X 0,Y 510.63,Z 579.366,A -85,B 0,C 180,E1 -5503.024,E2 -5503.024} C_VEL
LIN {X 0,Y 511.021,Z 567.54,A -85,B 0,C 180,E1 -5504.027,E2 -5504.027} C_VEL
LIN {X 0,Y 511.489,Z 556.074,A -85,B 0,C 180,E1 -5504.827,E2 -5504.827} C_VEL
LIN {X 0,Y 511.874,Z 542.719,A -85,B 0,C 180,E1 -5505.579,E2 -5505.579} C_VEL
LIN {X 0,Y 512.23,Z 530.584,A -85,B 0,C 180,E1 -5506.115,E2 -5506.115} C_VEL
LIN {X 0,Y 512.568,Z 516.605,A -85,B 0,C 180,E1 -5506.573,E2 -5506.573} C_VEL
LIN {X 0,Y 512.387,Z 512.025,A -85,B 0,C 180,E1 -5506.7,E2 -5506.7} C_VEL
LIN {X 0,Y 510.256,Z 499.864,A -85,B 0,C 180,E1 -5507.006,E2 -5507.006} C_VEL
LIN {X 0,Y 509.988,Z 497.498,A -85,B 0,C 180,E1 -5507.079,E2 -5507.079} C_VEL
LIN {X 0,Y 510.223,Z 482.722,A -85,B 0,C 180,E1 -5510.142,E2 -5510.142} C_VEL
LIN {X 0,Y 510.498,Z 468.629,A -85,B 0,C 180,E1 -5513.1,E2 -5513.1} C_VEL
LIN {X 0,Y 510.852,Z 453.519,A -85,B 0,C 180,E1 -5516.355,E2 -5516.355} C_VEL
LIN {X 0,Y 511.219,Z 438.623,A -85,B 0,C 180,E1 -5519.663,E2 -5519.663} C_VEL
LIN {X 0,Y 511.584,Z 425.23,A -85,B 0,C 180,E1 -5522.737,E2 -5522.737} C_VEL
LIN {X 0,Y 512.064,Z 410.774,A -85,B 0,C 180,E1 -5526.167,E2 -5526.167} C_VEL
LIN {X 0,Y 512.528,Z 400.057,A -85,B 0,C 180,E1 -5528.798,E2 -5528.798} C_VEL
LIN {X 0,Y 511.808,Z 394.759,A -85,B 0,C 180,E1 -5530.193,E2 -5530.193} C_VEL
LIN {X 0,Y 509.867,Z 385.599,A -85,B 0,C 180,E1 -5532.757,E2 -5532.757} C_VEL
LIN {X 0,Y 509.824,Z 385.607,A -85,B 0,C 180,E1 -5535.791,E2 -5535.791} C_VEL
LIN {X 0,Y 509.865,Z 385.597,A -85,B 0,C 180,E1 -5538.575,E2 -5538.575} C_VEL
LIN {X 0,Y 509.848,Z 385.605,A -85,B 0,C 180,E1 -5541.785,E2 -5541.785} C_VEL
LIN {X 0,Y 509.838,Z 385.599,A -85,B 0,C 180,E1 -5544.623,E2 -5544.623} C_VEL
LIN {X 0,Y 509.857,Z 385.603,A -85,B 0,C 180,E1 -5547.481,E2 -5547.481} C_VEL
LIN {X 0,Y 509.872,Z 385.597,A -85,B 0,C 180,E1 -5550.268,E2 -5550.268} C_VEL
LIN {X 0,Y 509.878,Z 385.595,A -85,B 0,C 180,E1 -5552.944,E2 -5552.944} C_VEL
LIN {X 0,Y 509.86,Z 385.602,A -85,B 0,C 180,E1 -5555.574,E2 -5555.574} C_VEL
LIN {X 0,Y 509.813,Z 385.605,A -85,B 0,C 180,E1 -5558.148,E2 -5558.148} C_VEL
LIN {X 0,Y 509.855,Z 385.597,A -85,B 0,C 180,E1 -5560.681,E2 -5560.681} C_VEL
LIN {X 0,Y 509.877,Z 385.598,A -85,B 0,C 180,E1 -5563.175,E2 -5563.175} C_VEL
LIN {X 0,Y 509.863,Z 385.601,A -85,B 0,C 180,E1 -5565.634,E2 -5565.634} C_VEL
LIN {X 0,Y 509.915,Z 385.591,A -85,B 0,C 180,E1 -5568.875,E2 -5568.875} C_VEL
LIN {X 0,Y 509.941,Z 385.588,A -85,B 0,C 180,E1 -5572.078,E2 -5572.078} C_VEL
LIN {X 0,Y 509.974,Z 385.582,A -85,B 0,C 180,E1 -5574.464,E2 -5574.464} C_VEL
LIN {X 0,Y 510.046,Z 385.577,A -85,B 0,C 180,E1 -5577.631,E2 -5577.631} C_VEL
LIN {X 0,Y 510.056,Z 385.573,A -85,B 0,C 180,E1 -5580.79,E2 -5580.79} C_VEL
LIN {X 0,Y 509.95,Z 385.59,A -85,B 0,C 180,E1 -5583.16,E2 -5583.16} C_VEL
LIN {X 0,Y 509.968,Z 385.583,A -85,B 0,C 180,E1 -5586.33,E2 -5586.33} C_VEL
LIN {X 0,Y 509.909,Z 385.591,A -85,B 0,C 180,E1 -5588.721,E2 -5588.721} C_VEL
LIN {X 0,Y 509.941,Z 385.588,A -85,B 0,C 180,E1 -5591.931,E2 -5591.931} C_VEL
LIN {X 0,Y 509.883,Z 385.6,A -85,B 0,C 180,E1 -5595.242,E2 -5595.242} C_VEL
LIN {X 0,Y 509.879,Z 385.595,A -85,B 0,C 180,E1 -5598.002,E2 -5598.002} C_VEL
LIN {X 0,Y 509.842,Z 385.603,A -85,B 0,C 180,E1 -5601.002,E2 -5601.002} C_VEL
LIN {X 0,Y 509.828,Z 385.604,A -85,B 0,C 180,E1 -5603.564,E2 -5603.564} C_VEL
LIN {X 0,Y 509.905,Z 385.591,A -85,B 0,C 180,E1 -5606.38,E2 -5606.38} C_VEL
LIN {X 0,Y 509.869,Z 385.599,A -85,B 0,C 180,E1 -5608.845,E2 -5608.845} C_VEL
LIN {X 0,Y 509.818,Z 385.605,A -85,B 0,C 180,E1 -5611.591,E2 -5611.591} C_VEL
LIN {X 0,Y 509.848,Z 385.599,A -85,B 0,C 180,E1 -5614.414,E2 -5614.414} C_VEL
LIN {X 0,Y 509.813,Z 385.606,A -85,B 0,C 180,E1 -5617.342,E2 -5617.342} C_VEL
LIN {X 0,Y 509.833,Z 385.6,A -85,B 0,C 180,E1 -5620.383,E2 -5620.383} C_VEL
LIN {X 0,Y 509.835,Z 385.605,A -85,B 0,C 180,E1 -5623.066,E2 -5623.066} C_VEL
LIN {X 0,Y 509.826,Z 385.602,A -85,B 0,C 180,E1 -5625.793,E2 -5625.793} C_VEL
LIN {X 0,Y 509.862,Z 385.598,A -85,B 0,C 180,E1 -5628.577,E2 -5628.577} C_VEL
LIN {X 0,Y 509.856,Z 385.599,A -85,B 0,C 180,E1 -5631.664,E2 -5631.664} C_VEL
LIN {X 0,Y 509.829,Z 385.602,A -85,B 0,C 180,E1 -5633.749,E2 -5633.749} C_VEL
LIN {X 0,Y 509.164,Z 385.685,A -85,B 0,C 180,E1 -5634.408,E2 -5634.408} C_VEL
LIN {X 0,Y 506.346,Z 386.038,A -85,B 0,C 180,E1 -5635.48,E2 -5635.48} C_VEL
LIN {X 0,Y 503.952,Z 386.339,A -85,B 0,C 180,E1 -5636.344,E2 -5636.344} C_VEL
LIN {X 0,Y 502.904,Z 386.468,A -85,B 0,C 180,E1 -5637.01,E2 -5637.01} C_VEL
LIN {X 0,Y 502.807,Z 386.477,A -85,B 0,C 180,E1 -5637.236,E2 -5637.236} C_VEL
LIN {X 0,Y 502.814,Z 386.475,A -85,B 0,C 180,E1 -5640.066,E2 -5640.066} C_VEL
LIN {X 0,Y 502.834,Z 386.475,A -85,B 0,C 180,E1 -5642.535,E2 -5642.535} C_VEL
LIN {X 0,Y 502.827,Z 386.476,A -85,B 0,C 180,E1 -5645.3,E2 -5645.3} C_VEL
LIN {X 0,Y 502.781,Z 386.479,A -85,B 0,C 180,E1 -5647.828,E2 -5647.828} C_VEL
LIN {X 0,Y 502.826,Z 386.475,A -85,B 0,C 180,E1 -5650.401,E2 -5650.401} C_VEL
LIN {X 0,Y 502.827,Z 386.477,A -85,B 0,C 180,E1 -5652.933,E2 -5652.933} C_VEL
LIN {X 0,Y 502.747,Z 386.487,A -85,B 0,C 180,E1 -5655.427,E2 -5655.427} C_VEL
LIN {X 0,Y 502.53,Z 386.516,A -85,B 0,C 180,E1 -5658.23,E2 -5658.23} C_VEL
LIN {X 0,Y 502.502,Z 386.521,A -85,B 0,C 180,E1 -5658.811,E2 -5658.811} C_VEL
LIN {X 0,Y 504.747,Z 395.218,A -85,B 0,C 180,E1 -5659.116,E2 -5659.116} C_VEL
LIN {X 0,Y 504.774,Z 407.654,A -85,B 0,C 180,E1 -5659.573,E2 -5659.573} C_VEL
LIN {X 0,Y 504.506,Z 419.731,A -85,B 0,C 180,E1 -5660.175,E2 -5660.175} C_VEL
LIN {X 0,Y 504.186,Z 430.495,A -85,B 0,C 180,E1 -5660.878,E2 -5660.878} C_VEL
LIN {X 0,Y 503.814,Z 441.488,A -85,B 0,C 180,E1 -5661.78,E2 -5661.78} C_VEL
LIN {X 0,Y 503.448,Z 451.286,A -85,B 0,C 180,E1 -5662.783,E2 -5662.783} C_VEL
LIN {X 0,Y 503.23,Z 460.632,A -85,B 0,C 180,E1 -5663.989,E2 -5663.989} C_VEL
LIN {X 0,Y 502.891,Z 468.185,A -85,B 0,C 180,E1 -5665.191,E2 -5665.191} C_VEL
LIN {X 0,Y 502.749,Z 474.195,A -85,B 0,C 180,E1 -5666.394,E2 -5666.394} C_VEL
LIN {X 0,Y 502.481,Z 478.992,A -85,B 0,C 180,E1 -5667.596,E2 -5667.596} C_VEL
LIN {X 0,Y 502.402,Z 482.672,A -85,B 0,C 180,E1 -5668.799,E2 -5668.799} C_VEL
LIN {X 0,Y 502.268,Z 485.382,A -85,B 0,C 180,E1 -5670.001,E2 -5670.001} C_VEL
LIN {X 0,Y 502.282,Z 487.539,A -85,B 0,C 180,E1 -5671.604,E2 -5671.604} C_VEL
LIN {X 0,Y 502.268,Z 488.059,A -85,B 0,C 180,E1 -5672.407,E2 -5672.407} C_VEL
LIN {X 0,Y 502.339,Z 487.87,A -85,B 0,C 180,E1 -5674.012,E2 -5674.012} C_VEL
LIN {X 0,Y 502.366,Z 486.186,A -85,B 0,C 180,E1 -5675.621,E2 -5675.621} C_VEL
LIN {X 0,Y 502.434,Z 482.836,A -85,B 0,C 180,E1 -5677.233,E2 -5677.233} C_VEL
LIN {X 0,Y 502.55,Z 479.171,A -85,B 0,C 180,E1 -5678.445,E2 -5678.445} C_VEL
LIN {X 0,Y 502.724,Z 474.394,A -85,B 0,C 180,E1 -5679.658,E2 -5679.658} C_VEL
LIN {X 0,Y 502.912,Z 468.357,A -85,B 0,C 180,E1 -5680.875,E2 -5680.875} C_VEL
LIN {X 0,Y 503.17,Z 460.598,A -85,B 0,C 180,E1 -5682.115,E2 -5682.115} C_VEL
LIN {X 0,Y 503.497,Z 451.229,A -85,B 0,C 180,E1 -5683.316,E2 -5683.316} C_VEL
LIN {X 0,Y 503.869,Z 441.234,A -85,B 0,C 180,E1 -5684.335,E2 -5684.335} C_VEL
LIN {X 0,Y 504.223,Z 429.984,A -85,B 0,C 180,E1 -5685.254,E2 -5685.254} C_VEL
LIN {X 0,Y 504.496,Z 419.648,A -85,B 0,C 180,E1 -5685.923,E2 -5685.923} C_VEL
LIN {X 0,Y 504.744,Z 407.334,A -85,B 0,C 180,E1 -5686.534,E2 -5686.534} C_VEL
LIN {X 0,Y 504.736,Z 395.203,A -85,B 0,C 180,E1 -5686.977,E2 -5686.977} C_VEL
LIN {X 0,Y 502.451,Z 386.527,A -85,B 0,C 180,E1 -5687.292,E2 -5687.292} C_VEL
LIN {X 0,Y 502.718,Z 386.491,A -85,B 0,C 180,E1 -5690.501,E2 -5690.501} C_VEL
LIN {X 0,Y 502.797,Z 386.482,A -85,B 0,C 180,E1 -5693.041,E2 -5693.041} C_VEL
LIN {X 0,Y 502.846,Z 386.471,A -85,B 0,C 180,E1 -5695.676,E2 -5695.676} C_VEL
LIN {X 0,Y 502.846,Z 386.472,A -85,B 0,C 180,E1 -5698.373,E2 -5698.373} C_VEL
LIN {X 0,Y 502.799,Z 386.478,A -85,B 0,C 180,E1 -5701.499,E2 -5701.499} C_VEL
LIN {X 0,Y 502.795,Z 386.478,A -85,B 0,C 180,E1 -5703.995,E2 -5703.995} C_VEL
LIN {X 0,Y 502.783,Z 386.476,A -85,B 0,C 180,E1 -5707.178,E2 -5707.178} C_VEL
LIN {X 0,Y 502.793,Z 386.476,A -85,B 0,C 180,E1 -5710.015,E2 -5710.015} C_VEL
LIN {X 0,Y 502.808,Z 386.479,A -85,B 0,C 180,E1 -5712.199,E2 -5712.199} C_VEL
LIN {X 0,Y 502.806,Z 386.473,A -85,B 0,C 180,E1 -5715.468,E2 -5715.468} C_VEL
LIN {X 0,Y 502.836,Z 386.474,A -85,B 0,C 180,E1 -5717.864,E2 -5717.864} C_VEL
LIN {X 0,Y 502.807,Z 386.462,A -85,B 0,C 180,E1 -5721.024,E2 -5721.024} C_VEL
LIN {X 0,Y 502.789,Z 386.483,A -85,B 0,C 180,E1 -5724.167,E2 -5724.167} C_VEL
LIN {X 0,Y 502.837,Z 386.469,A -85,B 0,C 180,E1 -5726.993,E2 -5726.993} C_VEL
LIN {X 0,Y 502.819,Z 386.462,A -85,B 0,C 180,E1 -5730.065,E2 -5730.065} C_VEL
LIN {X 0,Y 502.837,Z 386.466,A -85,B 0,C 180,E1 -5732.533,E2 -5732.533} C_VEL
LIN {X 0,Y 502.807,Z 386.477,A -85,B 0,C 180,E1 -5735.305,E2 -5735.305} C_VEL
LIN {X 0,Y 502.784,Z 386.483,A -85,B 0,C 180,E1 -5737.826,E2 -5737.826} C_VEL
LIN {X 0,Y 502.827,Z 386.472,A -85,B 0,C 180,E1 -5740.4,E2 -5740.4} C_VEL
LIN {X 0,Y 502.824,Z 386.476,A -85,B 0,C 180,E1 -5742.931,E2 -5742.931} C_VEL
LIN {X 0,Y 502.881,Z 386.627,A -85,B 0,C 180,E1 -5744.647,E2 -5744.647} C_VEL
LIN {X 0,Y 505.444,Z 395.206,A -85,B 0,C 180,E1 -5745.124,E2 -5745.124} C_VEL
LIN {X 0,Y 505.103,Z 407.724,A -85,B 0,C 180,E1 -5745.804,E2 -5745.804} C_VEL
LIN {X 0,Y 504.659,Z 419.653,A -85,B 0,C 180,E1 -5746.613,E2 -5746.613} C_VEL
LIN {X 0,Y 504.238,Z 430.994,A -85,B 0,C 180,E1 -5747.56,E2 -5747.56} C_VEL
LIN {X 0,Y 503.883,Z 440.712,A -85,B 0,C 180,E1 -5748.536,E2 -5748.536} C_VEL
LIN {X 0,Y 503.375,Z 450.796,A -85,B 0,C 180,E1 -5749.746,E2 -5749.746} C_VEL
LIN {X 0,Y 503.033,Z 460.313,A -85,B 0,C 180,E1 -5751.159,E2 -5751.159} C_VEL
LIN {X 0,Y 502.774,Z 466.995,A -85,B 0,C 180,E1 -5752.369,E2 -5752.369} C_VEL
LIN {X 0,Y 502.619,Z 472.564,A -85,B 0,C 180,E1 -5753.577,E2 -5753.577} C_VEL
LIN {X 0,Y 502.438,Z 477.12,A -85,B 0,C 180,E1 -5754.783,E2 -5754.783} C_VEL
LIN {X 0,Y 502.416,Z 480.716,A -85,B 0,C 180,E1 -5755.989,E2 -5755.989} C_VEL
LIN {X 0,Y 502.273,Z 484.311,A -85,B 0,C 180,E1 -5757.594,E2 -5757.594} C_VEL
LIN {X 0,Y 502.187,Z 486.533,A -85,B 0,C 180,E1 -5759.198,E2 -5759.198} C_VEL
LIN {X 0,Y 502.185,Z 487.432,A -85,B 0,C 180,E1 -5760.802,E2 -5760.802} C_VEL
LIN {X 0,Y 502.262,Z 487.015,A -85,B 0,C 180,E1 -5762.406,E2 -5762.406} C_VEL
LIN {X 0,Y 502.348,Z 485.34,A -85,B 0,C 180,E1 -5764.011,E2 -5764.011} C_VEL
LIN {X 0,Y 502.49,Z 482.316,A -85,B 0,C 180,E1 -5765.618,E2 -5765.618} C_VEL
LIN {X 0,Y 502.511,Z 479.216,A -85,B 0,C 180,E1 -5766.787,E2 -5766.787} C_VEL
LIN {X 0,Y 502.648,Z 475,A -85,B 0,C 180,E1 -5768.037,E2 -5768.037} C_VEL
LIN {X 0,Y 502.801,Z 469.964,A -85,B 0,C 180,E1 -5769.25,E2 -5769.25} C_VEL
LIN {X 0,Y 503.11,Z 462.656,A -85,B 0,C 180,E1 -5770.666,E2 -5770.666} C_VEL
LIN {X 0,Y 503.389,Z 455.019,A -85,B 0,C 180,E1 -5771.881,E2 -5771.881} C_VEL
LIN {X 0,Y 503.823,Z 445.696,A -85,B 0,C 180,E1 -5773.101,E2 -5773.101} C_VEL
LIN {X 0,Y 504.228,Z 435.342,A -85,B 0,C 180,E1 -5774.221,E2 -5774.221} C_VEL
LIN {X 0,Y 504.691,Z 423.845,A -85,B 0,C 180,E1 -5775.239,E2 -5775.239} C_VEL
LIN {X 0,Y 505.074,Z 412.548,A -85,B 0,C 180,E1 -5776.056,E2 -5776.056} C_VEL
LIN {X 0,Y 505.495,Z 400.319,A -85,B 0,C 180,E1 -5776.767,E2 -5776.767} C_VEL
LIN {X 0,Y 505.456,Z 395.11,A -85,B 0,C 180,E1 -5777.029,E2 -5777.029} C_VEL
LIN {X 0,Y 502.883,Z 386.471,A -85,B 0,C 180,E1 -5777.512,E2 -5777.512} C_VEL
LIN {X 0,Y 502.832,Z 386.479,A -85,B 0,C 180,E1 -5780.536,E2 -5780.536} C_VEL
LIN {X 0,Y 502.8,Z 386.484,A -85,B 0,C 180,E1 -5783.04,E2 -5783.04} C_VEL
LIN {X 0,Y 502.843,Z 386.477,A -85,B 0,C 180,E1 -5785.675,E2 -5785.675} C_VEL
LIN {X 0,Y 502.843,Z 386.474,A -85,B 0,C 180,E1 -5788.372,E2 -5788.372} C_VEL
LIN {X 0,Y 502.797,Z 386.483,A -85,B 0,C 180,E1 -5791.499,E2 -5791.499} C_VEL
LIN {X 0,Y 502.806,Z 386.481,A -85,B 0,C 180,E1 -5793.994,E2 -5793.994} C_VEL
LIN {X 0,Y 502.78,Z 386.483,A -85,B 0,C 180,E1 -5797.177,E2 -5797.177} C_VEL
LIN {X 0,Y 502.791,Z 386.483,A -85,B 0,C 180,E1 -5800.015,E2 -5800.015} C_VEL
LIN {X 0,Y 502.806,Z 386.48,A -85,B 0,C 180,E1 -5802.199,E2 -5802.199} C_VEL
LIN {X 0,Y 502.804,Z 386.484,A -85,B 0,C 180,E1 -5805.468,E2 -5805.468} C_VEL
LIN {X 0,Y 502.823,Z 386.48,A -85,B 0,C 180,E1 -5808.934,E2 -5808.934} C_VEL
LIN {X 0,Y 502.817,Z 386.567,A -85,B 0,C 180,E1 -5809.396,E2 -5809.396} C_VEL
LIN {X 0,Y 504.047,Z 393.31,A -85,B 0,C 180,E1 -5811.335,E2 -5811.335} C_VEL
LIN {X 0,Y 503.82,Z 400.548,A -85,B 0,C 180,E1 -5813.142,E2 -5813.142} C_VEL
LIN {X 0,Y 503.372,Z 416.941,A -85,B 0,C 180,E1 -5816.899,E2 -5816.899} C_VEL
LIN {X 0,Y 503.38,Z 431.155,A -85,B 0,C 180,E1 -5819.954,E2 -5819.954} C_VEL
LIN {X 0,Y 503.289,Z 445.877,A -85,B 0,C 180,E1 -5822.99,E2 -5822.99} C_VEL
LIN {X 0,Y 503.228,Z 460.247,A -85,B 0,C 180,E1 -5825.889,E2 -5825.889} C_VEL
LIN {X 0,Y 503.105,Z 474.405,A -85,B 0,C 180,E1 -5828.702,E2 -5828.702} C_VEL
LIN {X 0,Y 502.968,Z 487.307,A -85,B 0,C 180,E1 -5831.253,E2 -5831.253} C_VEL
LIN {X 0,Y 502.885,Z 494.747,A -85,B 0,C 180,E1 -5832.723,E2 -5832.723} C_VEL
LIN {X 0,Y 504.208,Z 506.505,A -85,B 0,C 180,E1 -5832.986,E2 -5832.986} C_VEL
LIN {X 0,Y 505.638,Z 514.452,A -85,B 0,C 180,E1 -5833.229,E2 -5833.229} C_VEL
LIN {X 0,Y 505.214,Z 528.821,A -85,B 0,C 180,E1 -5833.71,E2 -5833.71} C_VEL
LIN {X 0,Y 504.747,Z 542.873,A -85,B 0,C 180,E1 -5834.348,E2 -5834.348} C_VEL
LIN {X 0,Y 504.362,Z 556.746,A -85,B 0,C 180,E1 -5835.164,E2 -5835.164} C_VEL
LIN {X 0,Y 503.88,Z 569.181,A -85,B 0,C 180,E1 -5836.077,E2 -5836.077} C_VEL
LIN {X 0,Y 503.472,Z 580.563,A -85,B 0,C 180,E1 -5837.094,E2 -5837.094} C_VEL
LIN {X 0,Y 503.151,Z 590.563,A -85,B 0,C 180,E1 -5838.162,E2 -5838.162} C_VEL
LIN {X 0,Y 502.852,Z 599.717,A -85,B 0,C 180,E1 -5839.327,E2 -5839.327} C_VEL
LIN {X 0,Y 502.627,Z 607.717,A -85,B 0,C 180,E1 -5840.543,E2 -5840.543} C_VEL
LIN {X 0,Y 502.396,Z 615.334,A -85,B 0,C 180,E1 -5841.958,E2 -5841.958} C_VEL
LIN {X 0,Y 502.255,Z 622.18,A -85,B 0,C 180,E1 -5843.572,E2 -5843.572} C_VEL
LIN {X 0,Y 502.22,Z 626.205,A -85,B 0,C 180,E1 -5844.78,E2 -5844.78} C_VEL
LIN {X 0,Y 502.187,Z 629.287,A -85,B 0,C 180,E1 -5845.987,E2 -5845.987} C_VEL
LIN {X 0,Y 502.106,Z 632.112,A -85,B 0,C 180,E1 -5847.593,E2 -5847.593} C_VEL
LIN {X 0,Y 502.018,Z 633.506,A -85,B 0,C 180,E1 -5849.197,E2 -5849.197} C_VEL
LIN {X 0,Y 502.017,Z 633.516,A -85,B 0,C 180,E1 -5850.801,E2 -5850.801} C_VEL
LIN {X 0,Y 502.102,Z 632.145,A -85,B 0,C 180,E1 -5852.406,E2 -5852.406} C_VEL
LIN {X 0,Y 502.152,Z 629.355,A -85,B 0,C 180,E1 -5854.012,E2 -5854.012} C_VEL
LIN {X 0,Y 502.233,Z 625.082,A -85,B 0,C 180,E1 -5855.62,E2 -5855.62} C_VEL
LIN {X 0,Y 502.281,Z 619.185,A -85,B 0,C 180,E1 -5857.233,E2 -5857.233} C_VEL
LIN {X 0,Y 502.451,Z 612.551,A -85,B 0,C 180,E1 -5858.647,E2 -5858.647} C_VEL
LIN {X 0,Y 502.677,Z 604.325,A -85,B 0,C 180,E1 -5860.064,E2 -5860.064} C_VEL
LIN {X 0,Y 503.033,Z 595.74,A -85,B 0,C 180,E1 -5861.279,E2 -5861.279} C_VEL
LIN {X 0,Y 503.336,Z 585.774,A -85,B 0,C 180,E1 -5862.457,E2 -5862.457} C_VEL
LIN {X 0,Y 503.735,Z 575.038,A -85,B 0,C 180,E1 -5863.513,E2 -5863.513} C_VEL
LIN {X 0,Y 504.14,Z 563.849,A -85,B 0,C 180,E1 -5864.428,E2 -5864.428} C_VEL
LIN {X 0,Y 504.662,Z 551.793,A -85,B 0,C 180,E1 -5865.239,E2 -5865.239} C_VEL
LIN {X 0,Y 505.125,Z 538.587,A -85,B 0,C 180,E1 -5865.948,E2 -5865.948} C_VEL
LIN {X 0,Y 505.471,Z 524.859,A -85,B 0,C 180,E1 -5866.513,E2 -5866.513} C_VEL
LIN {X 0,Y 505.569,Z 513.431,A -85,B 0,C 180,E1 -5866.869,E2 -5866.869} C_VEL
LIN {X 0,Y 503.319,Z 500.042,A -85,B 0,C 180,E1 -5867.224,E2 -5867.224} C_VEL
LIN {X 0,Y 502.92,Z 496.762,A -85,B 0,C 180,E1 -5867.3,E2 -5867.3} C_VEL
LIN {X 0,Y 503.159,Z 482.885,A -85,B 0,C 180,E1 -5870.223,E2 -5870.223} C_VEL
LIN {X 0,Y 503.427,Z 469.89,A -85,B 0,C 180,E1 -5873.009,E2 -5873.009} C_VEL
LIN {X 0,Y 503.766,Z 455.904,A -85,B 0,C 180,E1 -5876.068,E2 -5876.068} C_VEL
LIN {X 0,Y 504.137,Z 441.987,A -85,B 0,C 180,E1 -5879.203,E2 -5879.203} C_VEL
LIN {X 0,Y 504.573,Z 428.074,A -85,B 0,C 180,E1 -5882.427,E2 -5882.427} C_VEL
LIN {X 0,Y 504.95,Z 416.152,A -85,B 0,C 180,E1 -5885.281,E2 -5885.281} C_VEL
LIN {X 0,Y 505.577,Z 404.229,A -85,B 0,C 180,E1 -5888.212,E2 -5888.212} C_VEL
LIN {X 0,Y 505.533,Z 400.085,A -85,B 0,C 180,E1 -5889.272,E2 -5889.272} C_VEL
LIN {X 0,Y 503.866,Z 391.33,A -85,B 0,C 180,E1 -5891.685,E2 -5891.685} C_VEL
LIN {X 0,Y 502.801,Z 386.48,A -85,B 0,C 180,E1 -5893.092,E2 -5893.092} C_VEL
LIN {X 0,Y 502.783,Z 386.484,A -85,B 0,C 180,E1 -5895.661,E2 -5895.661} C_VEL
LIN {X 0,Y 502.832,Z 386.478,A -85,B 0,C 180,E1 -5897.864,E2 -5897.864} C_VEL
LIN {X 0,Y 502.814,Z 386.475,A -85,B 0,C 180,E1 -5901.025,E2 -5901.025} C_VEL
LIN {X 0,Y 502.778,Z 386.482,A -85,B 0,C 180,E1 -5904.166,E2 -5904.166} C_VEL
LIN {X 0,Y 502.824,Z 386.474,A -85,B 0,C 180,E1 -5906.992,E2 -5906.992} C_VEL
LIN {X 0,Y 502.821,Z 386.476,A -85,B 0,C 180,E1 -5910.061,E2 -5910.061} C_VEL
LIN {X 0,Y 502.826,Z 386.473,A -85,B 0,C 180,E1 -5912.533,E2 -5912.533} C_VEL
LIN {X 0,Y 502.819,Z 386.478,A -85,B 0,C 180,E1 -5915.298,E2 -5915.298} C_VEL
LIN {X 0,Y 502.783,Z 386.482,A -85,B 0,C 180,E1 -5917.827,E2 -5917.827} C_VEL
LIN {X 0,Y 502.815,Z 386.475,A -85,B 0,C 180,E1 -5920.4,E2 -5920.4} C_VEL
LIN {X 0,Y 502.826,Z 386.474,A -85,B 0,C 180,E1 -5922.932,E2 -5922.932} C_VEL
LIN {X 0,Y 502.841,Z 386.477,A -85,B 0,C 180,E1 -5925.429,E2 -5925.429} C_VEL
LIN {X 0,Y 502.884,Z 386.466,A -85,B 0,C 180,E1 -5928.717,E2 -5928.717} C_VEL
LIN {X 0,Y 502.892,Z 386.468,A -85,B 0,C 180,E1 -5931.967,E2 -5931.967} C_VEL
LIN {X 0,Y 502.929,Z 386.46,A -85,B 0,C 180,E1 -5934.387,E2 -5934.387} C_VEL
LIN {X 0,Y 503.015,Z 386.453,A -85,B 0,C 180,E1 -5937.598,E2 -5937.598} C_VEL
LIN {X 0,Y 503.016,Z 386.451,A -85,B 0,C 180,E1 -5940,E2 -5940} C_VEL
LIN {X 0,Y 503.015,Z 386.449,A -85,B 0,C 180,E1 -5942.402,E2 -5942.402} C_VEL
LIN {X 0,Y 502.938,Z 386.462,A -85,B 0,C 180,E1 -5945.614,E2 -5945.614} C_VEL
LIN {X 0,Y 502.892,Z 386.466,A -85,B 0,C 180,E1 -5948.034,E2 -5948.034} C_VEL
LIN {X 0,Y 502.885,Z 386.471,A -85,B 0,C 180,E1 -5951.283,E2 -5951.283} C_VEL
LIN {X 0,Y 502.835,Z 386.472,A -85,B 0,C 180,E1 -5954.571,E2 -5954.571} C_VEL
LIN {X 0,Y 502.852,Z 386.471,A -85,B 0,C 180,E1 -5957.908,E2 -5957.908} C_VEL
LIN {X 0,Y 502.819,Z 386.474,A -85,B 0,C 180,E1 -5960.537,E2 -5960.537} C_VEL
LIN {X 0,Y 502.788,Z 386.483,A -85,B 0,C 180,E1 -5963.041,E2 -5963.041} C_VEL
LIN {X 0,Y 502.833,Z 386.475,A -85,B 0,C 180,E1 -5965.676,E2 -5965.676} C_VEL
LIN {X 0,Y 502.832,Z 386.472,A -85,B 0,C 180,E1 -5968.374,E2 -5968.374} C_VEL
LIN {X 0,Y 502.789,Z 386.481,A -85,B 0,C 180,E1 -5971.501,E2 -5971.501} C_VEL
LIN {X 0,Y 502.8,Z 386.477,A -85,B 0,C 180,E1 -5974.446,E2 -5974.446} C_VEL
LIN {X 0,Y 502.775,Z 386.484,A -85,B 0,C 180,E1 -5977.18,E2 -5977.18} C_VEL
LIN {X 0,Y 502.783,Z 386.479,A -85,B 0,C 180,E1 -5980.016,E2 -5980.016} C_VEL
LIN {X 0,Y 502.797,Z 386.477,A -85,B 0,C 180,E1 -5982.2,E2 -5982.2} C_VEL
LIN {X 0,Y 502.796,Z 386.48,A -85,B 0,C 180,E1 -5985.469,E2 -5985.469} C_VEL
LIN {X 0,Y 502.823,Z 386.479,A -85,B 0,C 180,E1 -5989.005,E2 -5989.005} C_VEL
LIN {X 0,Y 502.794,Z 386.477,A -85,B 0,C 180,E1 -5992.048,E2 -5992.048} C_VEL
LIN {X 0,Y 502.808,Z 386.48,A -85,B 0,C 180,E1 -5995.036,E2 -5995.036} C_VEL
LIN {X 0,Y 502.807,Z 386.477,A -85,B 0,C 180,E1 -5997.236,E2 -5997.236} C_VEL
LIN {X 0,Y 502.108,Z 386.564,A -85,B 0,C 180,E1 -5997.904,E2 -5997.904} C_VEL
LIN {X 0,Y 499.243,Z 386.924,A -85,B 0,C 180,E1 -5998.99,E2 -5998.99} C_VEL
LIN {X 0,Y 496.847,Z 387.219,A -85,B 0,C 180,E1 -5999.865,E2 -5999.865} C_VEL
LIN {X 0,Y 495.83,Z 387.347,A -85,B 0,C 180,E1 -6000.541,E2 -6000.541} C_VEL
LIN {X 0,Y 495.753,Z 387.354,A -85,B 0,C 180,E1 -6000.769,E2 -6000.769} C_VEL
LIN {X 0,Y 495.791,Z 387.35,A -85,B 0,C 180,E1 -6003.933,E2 -6003.933} C_VEL
LIN {X 0,Y 495.761,Z 387.356,A -85,B 0,C 180,E1 -6007.14,E2 -6007.14} C_VEL
LIN {X 0,Y 495.772,Z 387.352,A -85,B 0,C 180,E1 -6010.111,E2 -6010.111} C_VEL
LIN {X 0,Y 495.781,Z 387.356,A -85,B 0,C 180,E1 -6012.682,E2 -6012.682} C_VEL
LIN {X 0,Y 495.719,Z 387.363,A -85,B 0,C 180,E1 -6015.216,E2 -6015.216} C_VEL
LIN {X 0,Y 495.509,Z 387.39,A -85,B 0,C 180,E1 -6018.142,E2 -6018.142} C_VEL
LIN {X 0,Y 495.494,Z 387.539,A -85,B 0,C 180,E1 -6018.619,E2 -6018.619} C_VEL
LIN {X 0,Y 497.98,Z 396.717,A -85,B 0,C 180,E1 -6018.94,E2 -6018.94} C_VEL
LIN {X 0,Y 497.933,Z 409.632,A -85,B 0,C 180,E1 -6019.428,E2 -6019.428} C_VEL
LIN {X 0,Y 497.638,Z 421.412,A -85,B 0,C 180,E1 -6020.039,E2 -6020.039} C_VEL
LIN {X 0,Y 497.258,Z 433.393,A -85,B 0,C 180,E1 -6020.852,E2 -6020.852} C_VEL
LIN {X 0,Y 496.897,Z 444.018,A -85,B 0,C 180,E1 -6021.768,E2 -6021.768} C_VEL
LIN {X 0,Y 496.448,Z 454.329,A -85,B 0,C 180,E1 -6022.885,E2 -6022.885} C_VEL
LIN {X 0,Y 496.29,Z 461.922,A -85,B 0,C 180,E1 -6023.904,E2 -6023.904} C_VEL
LIN {X 0,Y 495.922,Z 469.416,A -85,B 0,C 180,E1 -6025.123,E2 -6025.123} C_VEL
LIN {X 0,Y 495.767,Z 475.374,A -85,B 0,C 180,E1 -6026.343,E2 -6026.343} C_VEL
LIN {X 0,Y 495.482,Z 480.134,A -85,B 0,C 180,E1 -6027.562,E2 -6027.562} C_VEL
LIN {X 0,Y 495.411,Z 483.777,A -85,B 0,C 180,E1 -6028.782,E2 -6028.782} C_VEL
LIN {X 0,Y 495.271,Z 486.453,A -85,B 0,C 180,E1 -6030.001,E2 -6030.001} C_VEL
LIN {X 0,Y 495.271,Z 488.581,A -85,B 0,C 180,E1 -6031.627,E2 -6031.627} C_VEL
LIN {X 0,Y 495.241,Z 489.076,A -85,B 0,C 180,E1 -6032.441,E2 -6032.441} C_VEL
LIN {X 0,Y 495.312,Z 488.851,A -85,B 0,C 180,E1 -6034.069,E2 -6034.069} C_VEL
LIN {X 0,Y 495.342,Z 488.187,A -85,B 0,C 180,E1 -6034.884,E2 -6034.884} C_VEL
LIN {X 0,Y 495.357,Z 487.117,A -85,B 0,C 180,E1 -6035.7,E2 -6035.7} C_VEL
LIN {X 0,Y 495.448,Z 483.731,A -85,B 0,C 180,E1 -6037.336,E2 -6037.336} C_VEL
LIN {X 0,Y 495.577,Z 480.029,A -85,B 0,C 180,E1 -6038.564,E2 -6038.564} C_VEL
LIN {X 0,Y 495.772,Z 475.211,A -85,B 0,C 180,E1 -6039.795,E2 -6039.795} C_VEL
LIN {X 0,Y 495.969,Z 469.115,A -85,B 0,C 180,E1 -6041.029,E2 -6041.029} C_VEL
LIN {X 0,Y 496.24,Z 461.44,A -85,B 0,C 180,E1 -6042.266,E2 -6042.266} C_VEL
LIN {X 0,Y 496.544,Z 453.581,A -85,B 0,C 180,E1 -6043.298,E2 -6043.298} C_VEL
LIN {X 0,Y 496.922,Z 443.982,A -85,B 0,C 180,E1 -6044.331,E2 -6044.331} C_VEL
LIN {X 0,Y 497.265,Z 433.133,A -85,B 0,C 180,E1 -6045.263,E2 -6045.263} C_VEL
LIN {X 0,Y 497.625,Z 422.295,A -85,B 0,C 180,E1 -6046.001,E2 -6046.001} C_VEL
LIN {X 0,Y 497.864,Z 410.867,A -85,B 0,C 180,E1 -6046.611,E2 -6046.611} C_VEL
LIN {X 0,Y 498.043,Z 398.101,A -85,B 0,C 180,E1 -6047.106,E2 -6047.106} C_VEL
LIN {X 0,Y 497.272,Z 393.669,A -85,B 0,C 180,E1 -6047.266,E2 -6047.266} C_VEL
LIN {X 0,Y 495.418,Z 387.402,A -85,B 0,C 180,E1 -6047.484,E2 -6047.484} C_VEL
LIN {X 0,Y 495.682,Z 387.368,A -85,B 0,C 180,E1 -6050.761,E2 -6050.761} C_VEL
LIN {X 0,Y 495.754,Z 387.357,A -85,B 0,C 180,E1 -6053.388,E2 -6053.388} C_VEL
LIN {X 0,Y 495.797,Z 387.348,A -85,B 0,C 180,E1 -6056.068,E2 -6056.068} C_VEL
LIN {X 0,Y 495.779,Z 387.357,A -85,B 0,C 180,E1 -6058.815,E2 -6058.815} C_VEL
LIN {X 0,Y 495.761,Z 387.354,A -85,B 0,C 180,E1 -6061.725,E2 -6061.725} C_VEL
LIN {X 0,Y 495.769,Z 387.359,A -85,B 0,C 180,E1 -6064.693,E2 -6064.693} C_VEL
LIN {X 0,Y 495.734,Z 387.352,A -85,B 0,C 180,E1 -6067.562,E2 -6067.562} C_VEL
LIN {X 0,Y 495.772,Z 387.357,A -85,B 0,C 180,E1 -6070.7,E2 -6070.7} C_VEL
LIN {X 0,Y 495.74,Z 387.357,A -85,B 0,C 180,E1 -6074.001,E2 -6074.001} C_VEL
LIN {X 0,Y 495.739,Z 387.355,A -85,B 0,C 180,E1 -6077.118,E2 -6077.118} C_VEL
LIN {X 0,Y 495.764,Z 387.353,A -85,B 0,C 180,E1 -6079.953,E2 -6079.953} C_VEL
LIN {X 0,Y 495.736,Z 387.354,A -85,B 0,C 180,E1 -6082.553,E2 -6082.553} C_VEL
LIN {X 0,Y 495.788,Z 387.35,A -85,B 0,C 180,E1 -6085.457,E2 -6085.457} C_VEL
LIN {X 0,Y 495.76,Z 387.346,A -85,B 0,C 180,E1 -6088.364,E2 -6088.364} C_VEL
LIN {X 0,Y 495.792,Z 387.337,A -85,B 0,C 180,E1 -6091.507,E2 -6091.507} C_VEL
LIN {X 0,Y 495.785,Z 387.354,A -85,B 0,C 180,E1 -6093.931,E2 -6093.931} C_VEL
LIN {X 0,Y 495.763,Z 387.354,A -85,B 0,C 180,E1 -6097.139,E2 -6097.139} C_VEL
LIN {X 0,Y 495.774,Z 387.353,A -85,B 0,C 180,E1 -6100.109,E2 -6100.109} C_VEL
LIN {X 0,Y 495.769,Z 387.353,A -85,B 0,C 180,E1 -6102.68,E2 -6102.68} C_VEL
LIN {X 0,Y 495.812,Z 387.469,A -85,B 0,C 180,E1 -6104.419,E2 -6104.419} C_VEL
LIN {X 0,Y 498.621,Z 397.336,A -85,B 0,C 180,E1 -6104.977,E2 -6104.977} C_VEL
LIN {X 0,Y 498.2,Z 410.196,A -85,B 0,C 180,E1 -6105.707,E2 -6105.707} C_VEL
LIN {X 0,Y 497.72,Z 423.079,A -85,B 0,C 180,E1 -6106.631,E2 -6106.631} C_VEL
LIN {X 0,Y 497.314,Z 433.84,A -85,B 0,C 180,E1 -6107.576,E2 -6107.576} C_VEL
LIN {X 0,Y 496.804,Z 443.412,A -85,B 0,C 180,E1 -6108.577,E2 -6108.577} C_VEL
LIN {X 0,Y 496.367,Z 453.162,A -85,B 0,C 180,E1 -6109.805,E2 -6109.805} C_VEL
LIN {X 0,Y 496.089,Z 461.232,A -85,B 0,C 180,E1 -6111.035,E2 -6111.035} C_VEL
LIN {X 0,Y 495.808,Z 467.951,A -85,B 0,C 180,E1 -6112.261,E2 -6112.261} C_VEL
LIN {X 0,Y 495.638,Z 473.541,A -85,B 0,C 180,E1 -6113.486,E2 -6113.486} C_VEL
LIN {X 0,Y 495.394,Z 479.412,A -85,B 0,C 180,E1 -6115.117,E2 -6115.117} C_VEL
LIN {X 0,Y 495.328,Z 483.706,A -85,B 0,C 180,E1 -6116.746,E2 -6116.746} C_VEL
LIN {X 0,Y 495.232,Z 486.596,A -85,B 0,C 180,E1 -6118.373,E2 -6118.373} C_VEL
LIN {X 0,Y 495.161,Z 488.153,A -85,B 0,C 180,E1 -6120,E2 -6120} C_VEL
LIN {X 0,Y 495.225,Z 488.42,A -85,B 0,C 180,E1 -6121.626,E2 -6121.626} C_VEL
LIN {X 0,Y 495.285,Z 487.396,A -85,B 0,C 180,E1 -6123.254,E2 -6123.254} C_VEL
LIN {X 0,Y 495.339,Z 485.054,A -85,B 0,C 180,E1 -6124.883,E2 -6124.883} C_VEL
LIN {X 0,Y 495.469,Z 482.349,A -85,B 0,C 180,E1 -6126.107,E2 -6126.107} C_VEL
LIN {X 0,Y 495.675,Z 477.482,A -85,B 0,C 180,E1 -6127.741,E2 -6127.741} C_VEL
LIN {X 0,Y 495.768,Z 472.738,A -85,B 0,C 180,E1 -6128.971,E2 -6128.971} C_VEL
LIN {X 0,Y 496.067,Z 465.871,A -85,B 0,C 180,E1 -6130.407,E2 -6130.407} C_VEL
LIN {X 0,Y 496.445,Z 457.385,A -85,B 0,C 180,E1 -6131.835,E2 -6131.835} C_VEL
LIN {X 0,Y 496.888,Z 448.291,A -85,B 0,C 180,E1 -6133.079,E2 -6133.079} C_VEL
LIN {X 0,Y 497.296,Z 438.24,A -85,B 0,C 180,E1 -6134.214,E2 -6134.214} C_VEL
LIN {X 0,Y 497.809,Z 427.107,A -85,B 0,C 180,E1 -6135.245,E2 -6135.245} C_VEL
LIN {X 0,Y 498.275,Z 414.726,A -85,B 0,C 180,E1 -6136.178,E2 -6136.178} C_VEL
LIN {X 0,Y 498.691,Z 402.844,A -85,B 0,C 180,E1 -6136.897,E2 -6136.897} C_VEL
LIN {X 0,Y 498.689,Z 396.751,A -85,B 0,C 180,E1 -6137.214,E2 -6137.214} C_VEL
LIN {X 0,Y 495.835,Z 387.351,A -85,B 0,C 180,E1 -6137.769,E2 -6137.769} C_VEL
LIN {X 0,Y 495.777,Z 387.357,A -85,B 0,C 180,E1 -6140.756,E2 -6140.756} C_VEL
LIN {X 0,Y 495.756,Z 387.36,A -85,B 0,C 180,E1 -6143.387,E2 -6143.387} C_VEL
LIN {X 0,Y 495.794,Z 387.354,A -85,B 0,C 180,E1 -6146.068,E2 -6146.068} C_VEL
LIN {X 0,Y 495.775,Z 387.355,A -85,B 0,C 180,E1 -6148.814,E2 -6148.814} C_VEL
LIN {X 0,Y 495.759,Z 387.358,A -85,B 0,C 180,E1 -6151.725,E2 -6151.725} C_VEL
LIN {X 0,Y 495.771,Z 387.356,A -85,B 0,C 180,E1 -6154.694,E2 -6154.694} C_VEL
LIN {X 0,Y 495.732,Z 387.363,A -85,B 0,C 180,E1 -6157.561,E2 -6157.561} C_VEL
LIN {X 0,Y 495.769,Z 387.357,A -85,B 0,C 180,E1 -6160.7,E2 -6160.7} C_VEL
LIN {X 0,Y 495.737,Z 387.364,A -85,B 0,C 180,E1 -6164.001,E2 -6164.001} C_VEL
LIN {X 0,Y 495.728,Z 387.365,A -85,B 0,C 180,E1 -6167.117,E2 -6167.117} C_VEL
LIN {X 0,Y 495.798,Z 387.422,A -85,B 0,C 180,E1 -6169.081,E2 -6169.081} C_VEL
LIN {X 0,Y 497.017,Z 393.998,A -85,B 0,C 180,E1 -6171.052,E2 -6171.052} C_VEL
LIN {X 0,Y 497.024,Z 399.718,A -85,B 0,C 180,E1 -6172.552,E2 -6172.552} C_VEL
LIN {X 0,Y 496.409,Z 415.237,A -85,B 0,C 180,E1 -6176.241,E2 -6176.241} C_VEL
LIN {X 0,Y 496.332,Z 428.188,A -85,B 0,C 180,E1 -6179.116,E2 -6179.116} C_VEL
LIN {X 0,Y 496.276,Z 440.655,A -85,B 0,C 180,E1 -6181.768,E2 -6181.768} C_VEL
LIN {X 0,Y 496.212,Z 456.362,A -85,B 0,C 180,E1 -6185.019,E2 -6185.019} C_VEL
LIN {X 0,Y 496.032,Z 471.879,A -85,B 0,C 180,E1 -6188.165,E2 -6188.165} C_VEL
LIN {X 0,Y 495.89,Z 485.863,A -85,B 0,C 180,E1 -6190.975,E2 -6190.975} C_VEL
LIN {X 0,Y 495.861,Z 493.323,A -85,B 0,C 180,E1 -6192.471,E2 -6192.471} C_VEL
LIN {X 0,Y 497.295,Z 507.412,A -85,B 0,C 180,E1 -6192.812,E2 -6192.812} C_VEL
LIN {X 0,Y 498.674,Z 515.486,A -85,B 0,C 180,E1 -6193.074,E2 -6193.074} C_VEL
LIN {X 0,Y 498.233,Z 530.385,A -85,B 0,C 180,E1 -6193.613,E2 -6193.613} C_VEL
LIN {X 0,Y 497.738,Z 543.272,A -85,B 0,C 180,E1 -6194.234,E2 -6194.234} C_VEL
LIN {X 0,Y 497.338,Z 556.637,A -85,B 0,C 180,E1 -6195.054,E2 -6195.054} C_VEL
LIN {X 0,Y 496.813,Z 568.875,A -85,B 0,C 180,E1 -6195.98,E2 -6195.98} C_VEL
LIN {X 0,Y 496.366,Z 581.145,A -85,B 0,C 180,E1 -6197.114,E2 -6197.114} C_VEL
LIN {X 0,Y 496.066,Z 590.874,A -85,B 0,C 180,E1 -6198.198,E2 -6198.198} C_VEL
LIN {X 0,Y 495.744,Z 599.804,A -85,B 0,C 180,E1 -6199.379,E2 -6199.379} C_VEL
LIN {X 0,Y 495.494,Z 608.789,A -85,B 0,C 180,E1 -6200.817,E2 -6200.817} C_VEL
LIN {X 0,Y 495.283,Z 616.027,A -85,B 0,C 180,E1 -6202.252,E2 -6202.252} C_VEL
LIN {X 0,Y 495.205,Z 621.963,A -85,B 0,C 180,E1 -6203.733,E2 -6203.733} C_VEL
LIN {X 0,Y 495.136,Z 626.2,A -85,B 0,C 180,E1 -6205.114,E2 -6205.114} C_VEL
LIN {X 0,Y 495.157,Z 628.204,A -85,B 0,C 180,E1 -6205.93,E2 -6205.93} C_VEL
LIN {X 0,Y 495.075,Z 631.064,A -85,B 0,C 180,E1 -6207.558,E2 -6207.558} C_VEL
LIN {X 0,Y 494.991,Z 632.484,A -85,B 0,C 180,E1 -6209.186,E2 -6209.186} C_VEL
LIN {X 0,Y 494.988,Z 632.512,A -85,B 0,C 180,E1 -6210.813,E2 -6210.813} C_VEL
LIN {X 0,Y 495.064,Z 631.15,A -85,B 0,C 180,E1 -6212.44,E2 -6212.44} C_VEL
LIN {X 0,Y 495.108,Z 628.365,A -85,B 0,C 180,E1 -6214.069,E2 -6214.069} C_VEL
LIN {X 0,Y 495.173,Z 624.089,A -85,B 0,C 180,E1 -6215.701,E2 -6215.701} C_VEL
LIN {X 0,Y 495.195,Z 620.019,A -85,B 0,C 180,E1 -6216.887,E2 -6216.887} C_VEL
LIN {X 0,Y 495.352,Z 613.629,A -85,B 0,C 180,E1 -6218.361,E2 -6218.361} C_VEL
LIN {X 0,Y 495.558,Z 605.843,A -85,B 0,C 180,E1 -6219.797,E2 -6219.797} C_VEL
LIN {X 0,Y 495.832,Z 597.752,A -85,B 0,C 180,E1 -6221.031,E2 -6221.031} C_VEL
LIN {X 0,Y 496.178,Z 588.004,A -85,B 0,C 180,E1 -6222.266,E2 -6222.266} C_VEL
LIN {X 0,Y 496.602,Z 577.238,A -85,B 0,C 180,E1 -6223.399,E2 -6223.399} C_VEL
LIN {X 0,Y 497.056,Z 565.375,A -85,B 0,C 180,E1 -6224.429,E2 -6224.429} C_VEL
LIN {X 0,Y 497.599,Z 553.871,A -85,B 0,C 180,E1 -6225.25,E2 -6225.25} C_VEL
LIN {X 0,Y 498.05,Z 541.483,A -85,B 0,C 180,E1 -6225.971,E2 -6225.971} C_VEL
LIN {X 0,Y 498.459,Z 528.428,A -85,B 0,C 180,E1 -6226.567,E2 -6226.567} C_VEL
LIN {X 0,Y 498.715,Z 514.637,A -85,B 0,C 180,E1 -6227.037,E2 -6227.037} C_VEL
LIN {X 0,Y 496.585,Z 501.445,A -85,B 0,C 180,E1 -6227.416,E2 -6227.416} C_VEL
LIN {X 0,Y 495.863,Z 495.903,A -85,B 0,C 180,E1 -6227.554,E2 -6227.554} C_VEL
LIN {X 0,Y 496.105,Z 482.095,A -85,B 0,C 180,E1 -6230.524,E2 -6230.524} C_VEL
LIN {X 0,Y 496.414,Z 469.172,A -85,B 0,C 180,E1 -6233.353,E2 -6233.353} C_VEL
LIN {X 0,Y 496.812,Z 455.253,A -85,B 0,C 180,E1 -6236.461,E2 -6236.461} C_VEL
LIN {X 0,Y 497.291,Z 439.637,A -85,B 0,C 180,E1 -6240.049,E2 -6240.049} C_VEL
LIN {X 0,Y 497.749,Z 425.48,A -85,B 0,C 180,E1 -6243.411,E2 -6243.411} C_VEL
LIN {X 0,Y 498.365,Z 411.441,A -85,B 0,C 180,E1 -6246.853,E2 -6246.853} C_VEL
LIN {X 0,Y 498.756,Z 403.933,A -85,B 0,C 180,E1 -6248.744,E2 -6248.744} C_VEL
LIN {X 0,Y 498.375,Z 399.809,A -85,B 0,C 180,E1 -6249.851,E2 -6249.851} C_VEL
LIN {X 0,Y 496.215,Z 389.306,A -85,B 0,C 180,E1 -6252.829,E2 -6252.829} C_VEL
LIN {X 0,Y 495.728,Z 387.363,A -85,B 0,C 180,E1 -6253.441,E2 -6253.441} C_VEL
LIN {X 0,Y 495.728,Z 387.359,A -85,B 0,C 180,E1 -6256.304,E2 -6256.304} C_VEL
LIN {X 0,Y 495.779,Z 387.354,A -85,B 0,C 180,E1 -6259.301,E2 -6259.301} C_VEL
LIN {X 0,Y 495.756,Z 387.358,A -85,B 0,C 180,E1 -6261.409,E2 -6261.409} C_VEL
LIN {X 0,Y 495.75,Z 387.355,A -85,B 0,C 180,E1 -6264.462,E2 -6264.462} C_VEL
LIN {X 0,Y 495.76,Z 387.358,A -85,B 0,C 180,E1 -6267.405,E2 -6267.405} C_VEL
LIN {X 0,Y 495.772,Z 387.353,A -85,B 0,C 180,E1 -6270.254,E2 -6270.254} C_VEL
LIN {X 0,Y 495.824,Z 387.349,A -85,B 0,C 180,E1 -6273.248,E2 -6273.248} C_VEL
LIN {X 0,Y 495.742,Z 387.359,A -85,B 0,C 180,E1 -6275.725,E2 -6275.725} C_VEL
LIN {X 0,Y 495.737,Z 387.357,A -85,B 0,C 180,E1 -6278.371,E2 -6278.371} C_VEL
LIN {X 0,Y 495.774,Z 387.353,A -85,B 0,C 180,E1 -6280.971,E2 -6280.971} C_VEL
LIN {X 0,Y 495.771,Z 387.357,A -85,B 0,C 180,E1 -6283.53,E2 -6283.53} C_VEL
LIN {X 0,Y 495.788,Z 387.352,A -85,B 0,C 180,E1 -6286.056,E2 -6286.056} C_VEL
LIN {X 0,Y 495.858,Z 387.341,A -85,B 0,C 180,E1 -6288.555,E2 -6288.555} C_VEL
LIN {X 0,Y 495.863,Z 387.343,A -85,B 0,C 180,E1 -6291.852,E2 -6291.852} C_VEL
LIN {X 0,Y 495.887,Z 387.338,A -85,B 0,C 180,E1 -6294.307,E2 -6294.307} C_VEL
LIN {X 0,Y 495.984,Z 387.329,A -85,B 0,C 180,E1 -6297.564,E2 -6297.564} C_VEL
LIN {X 0,Y 495.987,Z 387.327,A -85,B 0,C 180,E1 -6300,E2 -6300} C_VEL
LIN {X 0,Y 495.984,Z 387.325,A -85,B 0,C 180,E1 -6302.437,E2 -6302.437} C_VEL
LIN {X 0,Y 495.894,Z 387.339,A -85,B 0,C 180,E1 -6305.694,E2 -6305.694} C_VEL
LIN {X 0,Y 495.863,Z 387.341,A -85,B 0,C 180,E1 -6308.148,E2 -6308.148} C_VEL
LIN {X 0,Y 495.865,Z 387.344,A -85,B 0,C 180,E1 -6311.445,E2 -6311.445} C_VEL
LIN {X 0,Y 495.78,Z 387.353,A -85,B 0,C 180,E1 -6314.783,E2 -6314.783} C_VEL
LIN {X 0,Y 495.779,Z 387.355,A -85,B 0,C 180,E1 -6317.319,E2 -6317.319} C_VEL
LIN {X 0,Y 495.769,Z 387.354,A -85,B 0,C 180,E1 -6319.891,E2 -6319.891} C_VEL
LIN {X 0,Y 495.756,Z 387.357,A -85,B 0,C 180,E1 -6322.863,E2 -6322.863} C_VEL
LIN {X 0,Y 495.791,Z 387.35,A -85,B 0,C 180,E1 -6326.068,E2 -6326.068} C_VEL
LIN {X 0,Y 495.764,Z 387.356,A -85,B 0,C 180,E1 -6328.816,E2 -6328.816} C_VEL
LIN {X 0,Y 495.751,Z 387.357,A -85,B 0,C 180,E1 -6331.727,E2 -6331.727} C_VEL
LIN {X 0,Y 495.77,Z 387.354,A -85,B 0,C 180,E1 -6334.696,E2 -6334.696} C_VEL
LIN {X 0,Y 495.725,Z 387.36,A -85,B 0,C 180,E1 -6337.562,E2 -6337.562} C_VEL
LIN {X 0,Y 495.761,Z 387.356,A -85,B 0,C 180,E1 -6340.701,E2 -6340.701} C_VEL
LIN {X 0,Y 495.73,Z 387.359,A -85,B 0,C 180,E1 -6343.697,E2 -6343.697} C_VEL
LIN {X 0,Y 495.724,Z 387.358,A -85,B 0,C 180,E1 -6346.306,E2 -6346.306} C_VEL
LIN {X 0,Y 495.777,Z 387.354,A -85,B 0,C 180,E1 -6349.303,E2 -6349.303} C_VEL
LIN {X 0,Y 495.761,Z 387.356,A -85,B 0,C 180,E1 -6351.411,E2 -6351.411} C_VEL
LIN {X 0,Y 495.756,Z 387.355,A -85,B 0,C 180,E1 -6354.464,E2 -6354.464} C_VEL
LIN {X 0,Y 495.768,Z 387.355,A -85,B 0,C 180,E1 -6357.407,E2 -6357.407} C_VEL
LIN {X 0,Y 495.765,Z 387.353,A -85,B 0,C 180,E1 -6360.255,E2 -6360.255} C_VEL
LIN {X 0,Y 495.753,Z 387.354,A -85,B 0,C 180,E1 -6360.769,E2 -6360.769} C_VEL
LIN {X 0,Y 495.096,Z 387.439,A -85,B 0,C 180,E1 -6361.448,E2 -6361.448} C_VEL
LIN {X 0,Y 492.24,Z 387.795,A -85,B 0,C 180,E1 -6362.551,E2 -6362.551} C_VEL
LIN {X 0,Y 489.83,Z 388.095,A -85,B 0,C 180,E1 -6363.44,E2 -6363.44} C_VEL
LIN {X 0,Y 488.815,Z 388.219,A -85,B 0,C 180,E1 -6364.126,E2 -6364.126} C_VEL
LIN {X 0,Y 488.743,Z 388.229,A -85,B 0,C 180,E1 -6364.358,E2 -6364.358} C_VEL
LIN {X 0,Y 488.724,Z 388.233,A -85,B 0,C 180,E1 -6367.154,E2 -6367.154} C_VEL
LIN {X 0,Y 488.726,Z 388.23,A -85,B 0,C 180,E1 -6369.812,E2 -6369.812} C_VEL
LIN {X 0,Y 488.729,Z 388.232,A -85,B 0,C 180,E1 -6372.424,E2 -6372.424} C_VEL
LIN {X 0,Y 488.703,Z 388.237,A -85,B 0,C 180,E1 -6374.999,E2 -6374.999} C_VEL
LIN {X 0,Y 488.469,Z 388.268,A -85,B 0,C 180,E1 -6378.064,E2 -6378.064} C_VEL
LIN {X 0,Y 488.454,Z 388.361,A -85,B 0,C 180,E1 -6378.405,E2 -6378.405} C_VEL
LIN {X 0,Y 491.216,Z 398.206,A -85,B 0,C 180,E1 -6378.76,E2 -6378.76} C_VEL
LIN {X 0,Y 491.1,Z 410.413,A -85,B 0,C 180,E1 -6379.227,E2 -6379.227} C_VEL
LIN {X 0,Y 490.814,Z 421.419,A -85,B 0,C 180,E1 -6379.794,E2 -6379.794} C_VEL
LIN {X 0,Y 490.488,Z 432.248,A -85,B 0,C 180,E1 -6380.517,E2 -6380.517} C_VEL
LIN {X 0,Y 490.051,Z 443.289,A -85,B 0,C 180,E1 -6381.444,E2 -6381.444} C_VEL
LIN {X 0,Y 489.647,Z 452.915,A -85,B 0,C 180,E1 -6382.449,E2 -6382.449} C_VEL
LIN {X 0,Y 489.418,Z 461.798,A -85,B 0,C 180,E1 -6383.611,E2 -6383.611} C_VEL
LIN {X 0,Y 489.06,Z 469.491,A -85,B 0,C 180,E1 -6384.848,E2 -6384.848} C_VEL
LIN {X 0,Y 488.784,Z 474.727,A -85,B 0,C 180,E1 -6385.878,E2 -6385.878} C_VEL
LIN {X 0,Y 488.616,Z 479.825,A -85,B 0,C 180,E1 -6387.115,E2 -6387.115} C_VEL
LIN {X 0,Y 488.451,Z 483.794,A -85,B 0,C 180,E1 -6388.352,E2 -6388.352} C_VEL
LIN {X 0,Y 488.362,Z 485.891,A -85,B 0,C 180,E1 -6389.176,E2 -6389.176} C_VEL
LIN {X 0,Y 488.208,Z 488.769,A -85,B 0,C 180,E1 -6390.826,E2 -6390.826} C_VEL
LIN {X 0,Y 488.259,Z 489.623,A -85,B 0,C 180,E1 -6391.651,E2 -6391.651} C_VEL
LIN {X 0,Y 488.213,Z 490.089,A -85,B 0,C 180,E1 -6392.476,E2 -6392.476} C_VEL
LIN {X 0,Y 488.286,Z 489.832,A -85,B 0,C 180,E1 -6394.128,E2 -6394.128} C_VEL
LIN {X 0,Y 488.337,Z 489.149,A -85,B 0,C 180,E1 -6394.955,E2 -6394.955} C_VEL
LIN {X 0,Y 488.35,Z 488.047,A -85,B 0,C 180,E1 -6395.783,E2 -6395.783} C_VEL
LIN {X 0,Y 488.416,Z 486.058,A -85,B 0,C 180,E1 -6396.844,E2 -6396.844} C_VEL
LIN {X 0,Y 488.514,Z 482.258,A -85,B 0,C 180,E1 -6398.272,E2 -6398.272} C_VEL
LIN {X 0,Y 488.737,Z 477.769,A -85,B 0,C 180,E1 -6399.519,E2 -6399.519} C_VEL
LIN {X 0,Y 488.988,Z 470.985,A -85,B 0,C 180,E1 -6400.979,E2 -6400.979} C_VEL
LIN {X 0,Y 489.263,Z 464.073,A -85,B 0,C 180,E1 -6402.157,E2 -6402.157} C_VEL
LIN {X 0,Y 489.57,Z 455.936,A -85,B 0,C 180,E1 -6403.279,E2 -6403.279} C_VEL
LIN {X 0,Y 489.976,Z 446.602,A -85,B 0,C 180,E1 -6404.326,E2 -6404.326} C_VEL
LIN {X 0,Y 490.331,Z 436.243,A -85,B 0,C 180,E1 -6405.271,E2 -6405.271} C_VEL
LIN {X 0,Y 490.727,Z 424.654,A -85,B 0,C 180,E1 -6406.1,E2 -6406.1} C_VEL
LIN {X 0,Y 491.024,Z 412.012,A -85,B 0,C 180,E1 -6406.795,E2 -6406.795} C_VEL
LIN {X 0,Y 491.197,Z 399.601,A -85,B 0,C 180,E1 -6407.289,E2 -6407.289} C_VEL
LIN {X 0,Y 490.9,Z 396.718,A -85,B 0,C 180,E1 -6407.392,E2 -6407.392} C_VEL
LIN {X 0,Y 488.412,Z 388.274,A -85,B 0,C 180,E1 -6407.718,E2 -6407.718} C_VEL
LIN {X 0,Y 488.66,Z 388.244,A -85,B 0,C 180,E1 -6411.074,E2 -6411.074} C_VEL
LIN {X 0,Y 488.695,Z 388.234,A -85,B 0,C 180,E1 -6413.746,E2 -6413.746} C_VEL
LIN {X 0,Y 488.798,Z 388.226,A -85,B 0,C 180,E1 -6416.944,E2 -6416.944} C_VEL
LIN {X 0,Y 488.716,Z 388.233,A -85,B 0,C 180,E1 -6420.363,E2 -6420.363} C_VEL
LIN {X 0,Y 488.735,Z 388.23,A -85,B 0,C 180,E1 -6423.483,E2 -6423.483} C_VEL
LIN {X 0,Y 488.688,Z 388.239,A -85,B 0,C 180,E1 -6426.355,E2 -6426.355} C_VEL
LIN {X 0,Y 488.706,Z 388.23,A -85,B 0,C 180,E1 -6429.254,E2 -6429.254} C_VEL
LIN {X 0,Y 488.712,Z 388.23,A -85,B 0,C 180,E1 -6431.6,E2 -6431.6} C_VEL
LIN {X 0,Y 488.718,Z 388.23,A -85,B 0,C 180,E1 -6434.801,E2 -6434.801} C_VEL
LIN {X 0,Y 488.701,Z 388.232,A -85,B 0,C 180,E1 -6437.475,E2 -6437.475} C_VEL
LIN {X 0,Y 488.738,Z 388.226,A -85,B 0,C 180,E1 -6439.677,E2 -6439.677} C_VEL
LIN {X 0,Y 488.688,Z 388.229,A -85,B 0,C 180,E1 -6442.841,E2 -6442.841} C_VEL
LIN {X 0,Y 488.739,Z 388.233,A -85,B 0,C 180,E1 -6445.887,E2 -6445.887} C_VEL
LIN {X 0,Y 488.696,Z 388.222,A -85,B 0,C 180,E1 -6448.82,E2 -6448.82} C_VEL
LIN {X 0,Y 488.749,Z 388.215,A -85,B 0,C 180,E1 -6451.671,E2 -6451.671} C_VEL
LIN {X 0,Y 488.731,Z 388.228,A -85,B 0,C 180,E1 -6454.443,E2 -6454.443} C_VEL
LIN {X 0,Y 488.726,Z 388.231,A -85,B 0,C 180,E1 -6457.153,E2 -6457.153} C_VEL
LIN {X 0,Y 488.729,Z 388.234,A -85,B 0,C 180,E1 -6459.81,E2 -6459.81} C_VEL
LIN {X 0,Y 488.719,Z 388.231,A -85,B 0,C 180,E1 -6462.423,E2 -6462.423} C_VEL
LIN {X 0,Y 488.797,Z 388.419,A -85,B 0,C 180,E1 -6464.191,E2 -6464.191} C_VEL
LIN {X 0,Y 491.735,Z 398.069,A -85,B 0,C 180,E1 -6464.754,E2 -6464.754} C_VEL
LIN {X 0,Y 491.389,Z 411.043,A -85,B 0,C 180,E1 -6465.505,E2 -6465.505} C_VEL
LIN {X 0,Y 490.884,Z 423.928,A -85,B 0,C 180,E1 -6466.441,E2 -6466.441} C_VEL
LIN {X 0,Y 490.444,Z 434.711,A -85,B 0,C 180,E1 -6467.4,E2 -6467.4} C_VEL
LIN {X 0,Y 489.9,Z 444.29,A -85,B 0,C 180,E1 -6468.414,E2 -6468.414} C_VEL
LIN {X 0,Y 489.435,Z 454.058,A -85,B 0,C 180,E1 -6469.66,E2 -6469.66} C_VEL
LIN {X 0,Y 489.146,Z 462.148,A -85,B 0,C 180,E1 -6470.906,E2 -6470.906} C_VEL
LIN {X 0,Y 488.844,Z 468.898,A -85,B 0,C 180,E1 -6472.15,E2 -6472.15} C_VEL
LIN {X 0,Y 488.658,Z 474.509,A -85,B 0,C 180,E1 -6473.393,E2 -6473.393} C_VEL
LIN {X 0,Y 488.396,Z 480.389,A -85,B 0,C 180,E1 -6475.047,E2 -6475.047} C_VEL
LIN {X 0,Y 488.31,Z 484.701,A -85,B 0,C 180,E1 -6476.699,E2 -6476.699} C_VEL
LIN {X 0,Y 488.225,Z 487.606,A -85,B 0,C 180,E1 -6478.35,E2 -6478.35} C_VEL
LIN {X 0,Y 488.144,Z 489.187,A -85,B 0,C 180,E1 -6480,E2 -6480} C_VEL
LIN {X 0,Y 488.218,Z 489.452,A -85,B 0,C 180,E1 -6481.65,E2 -6481.65} C_VEL
LIN {X 0,Y 488.269,Z 488.434,A -85,B 0,C 180,E1 -6483.3,E2 -6483.3} C_VEL
LIN {X 0,Y 488.346,Z 486.091,A -85,B 0,C 180,E1 -6484.953,E2 -6484.953} C_VEL
LIN {X 0,Y 488.482,Z 483.374,A -85,B 0,C 180,E1 -6486.194,E2 -6486.194} C_VEL
LIN {X 0,Y 488.713,Z 478.498,A -85,B 0,C 180,E1 -6487.852,E2 -6487.852} C_VEL
LIN {X 0,Y 488.825,Z 473.731,A -85,B 0,C 180,E1 -6489.099,E2 -6489.099} C_VEL
LIN {X 0,Y 489.152,Z 466.839,A -85,B 0,C 180,E1 -6490.555,E2 -6490.555} C_VEL
LIN {X 0,Y 489.566,Z 458.315,A -85,B 0,C 180,E1 -6492.004,E2 -6492.004} C_VEL
LIN {X 0,Y 490.04,Z 449.176,A -85,B 0,C 180,E1 -6493.266,E2 -6493.266} C_VEL
LIN {X 0,Y 490.472,Z 439.093,A -85,B 0,C 180,E1 -6494.416,E2 -6494.416} C_VEL
LIN {X 0,Y 491.01,Z 427.927,A -85,B 0,C 180,E1 -6495.461,E2 -6495.461} C_VEL
LIN {X 0,Y 491.492,Z 415.686,A -85,B 0,C 180,E1 -6496.395,E2 -6496.395} C_VEL
LIN {X 0,Y 491.943,Z 403.532,A -85,B 0,C 180,E1 -6497.136,E2 -6497.136} C_VEL
LIN {X 0,Y 491.938,Z 398.462,A -85,B 0,C 180,E1 -6497.405,E2 -6497.405} C_VEL
LIN {X 0,Y 488.786,Z 388.228,A -85,B 0,C 180,E1 -6498.023,E2 -6498.023} C_VEL
LIN {X 0,Y 488.711,Z 388.237,A -85,B 0,C 180,E1 -6501.07,E2 -6501.07} C_VEL
LIN {X 0,Y 488.697,Z 388.239,A -85,B 0,C 180,E1 -6503.745,E2 -6503.745} C_VEL
LIN {X 0,Y 488.795,Z 388.225,A -85,B 0,C 180,E1 -6506.943,E2 -6506.943} C_VEL
LIN {X 0,Y 488.712,Z 388.236,A -85,B 0,C 180,E1 -6510.363,E2 -6510.363} C_VEL
LIN {X 0,Y 488.737,Z 388.231,A -85,B 0,C 180,E1 -6513.484,E2 -6513.484} C_VEL
LIN {X 0,Y 488.685,Z 388.24,A -85,B 0,C 180,E1 -6516.354,E2 -6516.354} C_VEL
LIN {X 0,Y 488.704,Z 388.238,A -85,B 0,C 180,E1 -6519.254,E2 -6519.254} C_VEL
LIN {X 0,Y 488.711,Z 388.237,A -85,B 0,C 180,E1 -6521.6,E2 -6521.6} C_VEL
LIN {X 0,Y 488.715,Z 388.238,A -85,B 0,C 180,E1 -6524.801,E2 -6524.801} C_VEL
LIN {X 0,Y 488.695,Z 388.241,A -85,B 0,C 180,E1 -6527.474,E2 -6527.474} C_VEL
LIN {X 0,Y 488.763,Z 388.412,A -85,B 0,C 180,E1 -6528.789,E2 -6528.789} C_VEL
LIN {X 0,Y 490.021,Z 395.103,A -85,B 0,C 180,E1 -6530.871,E2 -6530.871} C_VEL
LIN {X 0,Y 490.17,Z 399.409,A -85,B 0,C 180,E1 -6532.053,E2 -6532.053} C_VEL
LIN {X 0,Y 489.45,Z 412.089,A -85,B 0,C 180,E1 -6535.196,E2 -6535.196} C_VEL
LIN {X 0,Y 489.303,Z 424.917,A -85,B 0,C 180,E1 -6538.159,E2 -6538.159} C_VEL
LIN {X 0,Y 489.283,Z 438.707,A -85,B 0,C 180,E1 -6541.187,E2 -6541.187} C_VEL
LIN {X 0,Y 489.131,Z 454.194,A -85,B 0,C 180,E1 -6544.465,E2 -6544.465} C_VEL
LIN {X 0,Y 489.001,Z 468.313,A -85,B 0,C 180,E1 -6547.389,E2 -6547.389} C_VEL
LIN {X 0,Y 488.862,Z 484.45,A -85,B 0,C 180,E1 -6550.691,E2 -6550.691} C_VEL
LIN {X 0,Y 488.744,Z 491.891,A -85,B 0,C 180,E1 -6552.207,E2 -6552.207} C_VEL
LIN {X 0,Y 490.49,Z 508.948,A -85,B 0,C 180,E1 -6552.653,E2 -6552.653} C_VEL
LIN {X 0,Y 491.718,Z 516.922,A -85,B 0,C 180,E1 -6552.935,E2 -6552.935} C_VEL
LIN {X 0,Y 491.254,Z 531.137,A -85,B 0,C 180,E1 -6553.489,E2 -6553.489} C_VEL
LIN {X 0,Y 490.707,Z 545.135,A -85,B 0,C 180,E1 -6554.209,E2 -6554.209} C_VEL
LIN {X 0,Y 490.26,Z 558.002,A -85,B 0,C 180,E1 -6555.046,E2 -6555.046} C_VEL
LIN {X 0,Y 489.725,Z 569.814,A -85,B 0,C 180,E1 -6555.984,E2 -6555.984} C_VEL
LIN {X 0,Y 489.271,Z 581.762,A -85,B 0,C 180,E1 -6557.135,E2 -6557.135} C_VEL
LIN {X 0,Y 488.97,Z 592.461,A -85,B 0,C 180,E1 -6558.391,E2 -6558.391} C_VEL
LIN {X 0,Y 488.584,Z 601.313,A -85,B 0,C 180,E1 -6559.641,E2 -6559.641} C_VEL
LIN {X 0,Y 488.402,Z 608.726,A -85,B 0,C 180,E1 -6560.892,E2 -6560.892} C_VEL
LIN {X 0,Y 488.236,Z 614.837,A -85,B 0,C 180,E1 -6562.139,E2 -6562.139} C_VEL
LIN {X 0,Y 488.162,Z 621.049,A -85,B 0,C 180,E1 -6563.703,E2 -6563.703} C_VEL
LIN {X 0,Y 488.115,Z 625.103,A -85,B 0,C 180,E1 -6565.043,E2 -6565.043} C_VEL
LIN {X 0,Y 488.127,Z 627.123,A -85,B 0,C 180,E1 -6565.871,E2 -6565.871} C_VEL
LIN {X 0,Y 488.043,Z 630.016,A -85,B 0,C 180,E1 -6567.523,E2 -6567.523} C_VEL
LIN {X 0,Y 487.963,Z 631.462,A -85,B 0,C 180,E1 -6569.174,E2 -6569.174} C_VEL
LIN {X 0,Y 488.002,Z 631.667,A -85,B 0,C 180,E1 -6569.999,E2 -6569.999} C_VEL
LIN {X 0,Y 487.988,Z 631.007,A -85,B 0,C 180,E1 -6571.65,E2 -6571.65} C_VEL
LIN {X 0,Y 488.049,Z 628.946,A -85,B 0,C 180,E1 -6573.301,E2 -6573.301} C_VEL
LIN {X 0,Y 488.106,Z 625.431,A -85,B 0,C 180,E1 -6574.955,E2 -6574.955} C_VEL
LIN {X 0,Y 488.138,Z 620.356,A -85,B 0,C 180,E1 -6576.613,E2 -6576.613} C_VEL
LIN {X 0,Y 488.257,Z 613.591,A -85,B 0,C 180,E1 -6578.275,E2 -6578.275} C_VEL
LIN {X 0,Y 488.454,Z 606.064,A -85,B 0,C 180,E1 -6579.732,E2 -6579.732} C_VEL
LIN {X 0,Y 488.789,Z 596.721,A -85,B 0,C 180,E1 -6581.192,E2 -6581.192} C_VEL
LIN {X 0,Y 489.149,Z 586.957,A -85,B 0,C 180,E1 -6582.445,E2 -6582.445} C_VEL
LIN {X 0,Y 489.592,Z 576.173,A -85,B 0,C 180,E1 -6583.594,E2 -6583.594} C_VEL
LIN {X 0,Y 490.094,Z 564.305,A -85,B 0,C 180,E1 -6584.639,E2 -6584.639} C_VEL
LIN {X 0,Y 490.661,Z 552.782,A -85,B 0,C 180,E1 -6585.471,E2 -6585.471} C_VEL
LIN {X 0,Y 491.134,Z 540.991,A -85,B 0,C 180,E1 -6586.169,E2 -6586.169} C_VEL
LIN {X 0,Y 491.589,Z 527.317,A -85,B 0,C 180,E1 -6586.806,E2 -6586.806} C_VEL
LIN {X 0,Y 491.841,Z 515.57,A -85,B 0,C 180,E1 -6587.219,E2 -6587.219} C_VEL
LIN {X 0,Y 489.793,Z 502.442,A -85,B 0,C 180,E1 -6587.623,E2 -6587.623} C_VEL
LIN {X 0,Y 488.812,Z 495.181,A -85,B 0,C 180,E1 -6587.789,E2 -6587.789} C_VEL
LIN {X 0,Y 489.101,Z 480.311,A -85,B 0,C 180,E1 -6591.052,E2 -6591.052} C_VEL
LIN {X 0,Y 489.392,Z 468.45,A -85,B 0,C 180,E1 -6593.708,E2 -6593.708} C_VEL
LIN {X 0,Y 489.791,Z 454.891,A -85,B 0,C 180,E1 -6596.798,E2 -6596.798} C_VEL
LIN {X 0,Y 490.316,Z 440.709,A -85,B 0,C 180,E1 -6600.11,E2 -6600.11} C_VEL
LIN {X 0,Y 490.772,Z 426.989,A -85,B 0,C 180,E1 -6603.414,E2 -6603.414} C_VEL
LIN {X 0,Y 491.455,Z 412.903,A -85,B 0,C 180,E1 -6606.912,E2 -6606.912} C_VEL
LIN {X 0,Y 491.833,Z 404.956,A -85,B 0,C 180,E1 -6608.955,E2 -6608.955} C_VEL
LIN {X 0,Y 491.18,Z 399.849,A -85,B 0,C 180,E1 -6610.354,E2 -6610.354} C_VEL
LIN {X 0,Y 489.345,Z 391.013,A -85,B 0,C 180,E1 -6612.907,E2 -6612.907} C_VEL
LIN {X 0,Y 488.698,Z 388.239,A -85,B 0,C 180,E1 -6613.79,E2 -6613.79} C_VEL
LIN {X 0,Y 488.738,Z 388.23,A -85,B 0,C 180,E1 -6617.168,E2 -6617.168} C_VEL
LIN {X 0,Y 488.761,Z 388.232,A -85,B 0,C 180,E1 -6619.679,E2 -6619.679} C_VEL
LIN {X 0,Y 488.675,Z 388.236,A -85,B 0,C 180,E1 -6622.841,E2 -6622.841} C_VEL
LIN {X 0,Y 488.726,Z 388.232,A -85,B 0,C 180,E1 -6625.887,E2 -6625.887} C_VEL
LIN {X 0,Y 488.687,Z 388.235,A -85,B 0,C 180,E1 -6628.82,E2 -6628.82} C_VEL
LIN {X 0,Y 488.737,Z 388.232,A -85,B 0,C 180,E1 -6631.671,E2 -6631.671} C_VEL
LIN {X 0,Y 488.741,Z 388.228,A -85,B 0,C 180,E1 -6634.444,E2 -6634.444} C_VEL
LIN {X 0,Y 488.71,Z 388.234,A -85,B 0,C 180,E1 -6637.153,E2 -6637.153} C_VEL
LIN {X 0,Y 488.718,Z 388.233,A -85,B 0,C 180,E1 -6639.81,E2 -6639.81} C_VEL
LIN {X 0,Y 488.724,Z 388.23,A -85,B 0,C 180,E1 -6642.423,E2 -6642.423} C_VEL
LIN {X 0,Y 488.754,Z 388.228,A -85,B 0,C 180,E1 -6645,E2 -6645} C_VEL
LIN {X 0,Y 488.82,Z 388.218,A -85,B 0,C 180,E1 -6648.388,E2 -6648.388} C_VEL
LIN {X 0,Y 488.808,Z 388.222,A -85,B 0,C 180,E1 -6651.734,E2 -6651.734} C_VEL
LIN {X 0,Y 488.846,Z 388.216,A -85,B 0,C 180,E1 -6654.224,E2 -6654.224} C_VEL
LIN {X 0,Y 488.952,Z 388.205,A -85,B 0,C 180,E1 -6657.529,E2 -6657.529} C_VEL
LIN {X 0,Y 488.959,Z 388.203,A -85,B 0,C 180,E1 -6660,E2 -6660} C_VEL
LIN {X 0,Y 488.952,Z 388.202,A -85,B 0,C 180,E1 -6662.472,E2 -6662.472} C_VEL
LIN {X 0,Y 488.852,Z 388.216,A -85,B 0,C 180,E1 -6665.776,E2 -6665.776} C_VEL
LIN {X 0,Y 488.808,Z 388.22,A -85,B 0,C 180,E1 -6668.267,E2 -6668.267} C_VEL
LIN {X 0,Y 488.823,Z 388.22,A -85,B 0,C 180,E1 -6671.612,E2 -6671.612} C_VEL
LIN {X 0,Y 488.752,Z 388.23,A -85,B 0,C 180,E1 -6675.001,E2 -6675.001} C_VEL
LIN {X 0,Y 488.745,Z 388.228,A -85,B 0,C 180,E1 -6678.443,E2 -6678.443} C_VEL
LIN {X 0,Y 488.698,Z 388.239,A -85,B 0,C 180,E1 -6681.071,E2 -6681.071} C_VEL
LIN {X 0,Y 488.685,Z 388.237,A -85,B 0,C 180,E1 -6683.746,E2 -6683.746} C_VEL
LIN {X 0,Y 488.79,Z 388.226,A -85,B 0,C 180,E1 -6686.946,E2 -6686.946} C_VEL
LIN {X 0,Y 488.702,Z 388.233,A -85,B 0,C 180,E1 -6690.364,E2 -6690.364} C_VEL
LIN {X 0,Y 488.729,Z 388.232,A -85,B 0,C 180,E1 -6693.486,E2 -6693.486} C_VEL
LIN {X 0,Y 488.682,Z 388.236,A -85,B 0,C 180,E1 -6696.357,E2 -6696.357} C_VEL
LIN {X 0,Y 488.696,Z 388.237,A -85,B 0,C 180,E1 -6699.255,E2 -6699.255} C_VEL
LIN {X 0,Y 488.718,Z 388.233,A -85,B 0,C 180,E1 -6701.603,E2 -6701.603} C_VEL
LIN {X 0,Y 488.707,Z 388.236,A -85,B 0,C 180,E1 -6704.803,E2 -6704.803} C_VEL
LIN {X 0,Y 488.687,Z 388.237,A -85,B 0,C 180,E1 -6707.476,E2 -6707.476} C_VEL
LIN {X 0,Y 488.746,Z 388.231,A -85,B 0,C 180,E1 -6710.752,E2 -6710.752} C_VEL
LIN {X 0,Y 488.683,Z 388.236,A -85,B 0,C 180,E1 -6713.87,E2 -6713.87} C_VEL
LIN {X 0,Y 488.738,Z 388.233,A -85,B 0,C 180,E1 -6716.879,E2 -6716.879} C_VEL
LIN {X 0,Y 488.723,Z 388.231,A -85,B 0,C 180,E1 -6719.782,E2 -6719.782} C_VEL
LIN {X 0,Y 488.792,Z 388.225,A -85,B 0,C 180,E1 -6723.058,E2 -6723.058} C_VEL
LIN {X 0,Y 488.743,Z 388.229,A -85,B 0,C 180,E1 -6724.358,E2 -6724.358} C_VEL
LIN {X 0,Y 488.099,Z 388.313,A -85,B 0,C 180,E1 -6725.046,E2 -6725.046} C_VEL
LIN {X 0,Y 485.23,Z 388.67,A -85,B 0,C 180,E1 -6726.162,E2 -6726.162} C_VEL
LIN {X 0,Y 482.782,Z 388.973,A -85,B 0,C 180,E1 -6727.062,E2 -6727.062} C_VEL
LIN {X 0,Y 481.725,Z 389.103,A -85,B 0,C 180,E1 -6727.758,E2 -6727.758} C_VEL
LIN {X 0,Y 481.636,Z 389.113,A -85,B 0,C 180,E1 -6727.993,E2 -6727.993} C_VEL
LIN {X 0,Y 481.707,Z 389.106,A -85,B 0,C 180,E1 -6730.394,E2 -6730.394} C_VEL
LIN {X 0,Y 481.683,Z 389.11,A -85,B 0,C 180,E1 -6733.035,E2 -6733.035} C_VEL
LIN {X 0,Y 481.589,Z 389.123,A -85,B 0,C 180,E1 -6735.637,E2 -6735.637} C_VEL
LIN {X 0,Y 481.42,Z 389.146,A -85,B 0,C 180,E1 -6738.183,E2 -6738.183} C_VEL
LIN {X 0,Y 484.396,Z 399.61,A -85,B 0,C 180,E1 -6738.573,E2 -6738.573} C_VEL
LIN {X 0,Y 484.239,Z 412.302,A -85,B 0,C 180,E1 -6739.073,E2 -6739.073} C_VEL
LIN {X 0,Y 483.949,Z 423.065,A -85,B 0,C 180,E1 -6739.648,E2 -6739.648} C_VEL
LIN {X 0,Y 483.622,Z 433.764,A -85,B 0,C 180,E1 -6740.381,E2 -6740.381} C_VEL
LIN {X 0,Y 483.151,Z 444.725,A -85,B 0,C 180,E1 -6741.321,E2 -6741.321} C_VEL
LIN {X 0,Y 482.755,Z 453.999,A -85,B 0,C 180,E1 -6742.309,E2 -6742.309} C_VEL
LIN {X 0,Y 482.48,Z 463.083,A -85,B 0,C 180,E1 -6743.519,E2 -6743.519} C_VEL
LIN {X 0,Y 482.105,Z 470.73,A -85,B 0,C 180,E1 -6744.773,E2 -6744.773} C_VEL
LIN {X 0,Y 481.826,Z 475.922,A -85,B 0,C 180,E1 -6745.819,E2 -6745.819} C_VEL
LIN {X 0,Y 481.621,Z 480.985,A -85,B 0,C 180,E1 -6747.073,E2 -6747.073} C_VEL
LIN {X 0,Y 481.455,Z 484.918,A -85,B 0,C 180,E1 -6748.328,E2 -6748.328} C_VEL
LIN {X 0,Y 481.358,Z 486.984,A -85,B 0,C 180,E1 -6749.164,E2 -6749.164} C_VEL
LIN {X 0,Y 481.19,Z 489.827,A -85,B 0,C 180,E1 -6750.838,E2 -6750.838} C_VEL
LIN {X 0,Y 481.246,Z 490.664,A -85,B 0,C 180,E1 -6751.675,E2 -6751.675} C_VEL
LIN {X 0,Y 481.226,Z 491.14,A -85,B 0,C 180,E1 -6753.35,E2 -6753.35} C_VEL
LIN {X 0,Y 481.332,Z 490.107,A -85,B 0,C 180,E1 -6755.027,E2 -6755.027} C_VEL
LIN {X 0,Y 481.381,Z 487.453,A -85,B 0,C 180,E1 -6756.708,E2 -6756.708} C_VEL
LIN {X 0,Y 481.49,Z 484.365,A -85,B 0,C 180,E1 -6757.971,E2 -6757.971} C_VEL
LIN {X 0,Y 481.705,Z 480.22,A -85,B 0,C 180,E1 -6759.236,E2 -6759.236} C_VEL
LIN {X 0,Y 481.937,Z 474.907,A -85,B 0,C 180,E1 -6760.504,E2 -6760.504} C_VEL
LIN {X 0,Y 482.135,Z 468.248,A -85,B 0,C 180,E1 -6761.776,E2 -6761.776} C_VEL
LIN {X 0,Y 482.546,Z 459.83,A -85,B 0,C 180,E1 -6763.048,E2 -6763.048} C_VEL
LIN {X 0,Y 482.917,Z 451.188,A -85,B 0,C 180,E1 -6764.11,E2 -6764.11} C_VEL
LIN {X 0,Y 483.321,Z 441.679,A -85,B 0,C 180,E1 -6765.066,E2 -6765.066} C_VEL
LIN {X 0,Y 483.734,Z 431.148,A -85,B 0,C 180,E1 -6765.917,E2 -6765.917} C_VEL
LIN {X 0,Y 484.072,Z 419.225,A -85,B 0,C 180,E1 -6766.674,E2 -6766.674} C_VEL
LIN {X 0,Y 484.333,Z 407.224,A -85,B 0,C 180,E1 -6767.252,E2 -6767.252} C_VEL
LIN {X 0,Y 484.255,Z 398.711,A -85,B 0,C 180,E1 -6767.563,E2 -6767.563} C_VEL
LIN {X 0,Y 481.388,Z 389.149,A -85,B 0,C 180,E1 -6767.924,E2 -6767.924} C_VEL
LIN {X 0,Y 481.613,Z 389.12,A -85,B 0,C 180,E1 -6771.397,E2 -6771.397} C_VEL
LIN {X 0,Y 481.68,Z 389.107,A -85,B 0,C 180,E1 -6774.114,E2 -6774.114} C_VEL
LIN {X 0,Y 481.753,Z 389.103,A -85,B 0,C 180,E1 -6777.139,E2 -6777.139} C_VEL
LIN {X 0,Y 481.685,Z 389.107,A -85,B 0,C 180,E1 -6779.741,E2 -6779.741} C_VEL
LIN {X 0,Y 481.676,Z 389.114,A -85,B 0,C 180,E1 -6782.675,E2 -6782.675} C_VEL
LIN {X 0,Y 481.642,Z 389.113,A -85,B 0,C 180,E1 -6785.71,E2 -6785.71} C_VEL
LIN {X 0,Y 481.676,Z 389.108,A -85,B 0,C 180,E1 -6788.859,E2 -6788.859} C_VEL
LIN {X 0,Y 481.658,Z 389.111,A -85,B 0,C 180,E1 -6791.913,E2 -6791.913} C_VEL
LIN {X 0,Y 481.665,Z 389.114,A -85,B 0,C 180,E1 -6794.457,E2 -6794.457} C_VEL
LIN {X 0,Y 481.659,Z 389.111,A -85,B 0,C 180,E1 -6797.84,E2 -6797.84} C_VEL
LIN {X 0,Y 481.686,Z 389.094,A -85,B 0,C 180,E1 -6800.651,E2 -6800.651} C_VEL
LIN {X 0,Y 481.636,Z 389.108,A -85,B 0,C 180,E1 -6803.376,E2 -6803.376} C_VEL
LIN {X 0,Y 481.715,Z 389.104,A -85,B 0,C 180,E1 -6806.33,E2 -6806.33} C_VEL
LIN {X 0,Y 481.655,Z 389.101,A -85,B 0,C 180,E1 -6809.417,E2 -6809.417} C_VEL
LIN {X 0,Y 481.704,Z 389.1,A -85,B 0,C 180,E1 -6812.168,E2 -6812.168} C_VEL
LIN {X 0,Y 481.697,Z 389.104,A -85,B 0,C 180,E1 -6814.968,E2 -6814.968} C_VEL
LIN {X 0,Y 481.653,Z 389.117,A -85,B 0,C 180,E1 -6817.705,E2 -6817.705} C_VEL
LIN {X 0,Y 481.708,Z 389.104,A -85,B 0,C 180,E1 -6820.393,E2 -6820.393} C_VEL
LIN {X 0,Y 481.683,Z 389.111,A -85,B 0,C 180,E1 -6823.033,E2 -6823.033} C_VEL
LIN {X 0,Y 481.719,Z 389.107,A -85,B 0,C 180,E1 -6823.938,E2 -6823.938} C_VEL
LIN {X 0,Y 484.989,Z 399.946,A -85,B 0,C 180,E1 -6824.594,E2 -6824.594} C_VEL
